// TIA Portal V17 export
// export: Created 2023-12-05T13:40:23.3729222Z, ExportSetting WithDefaults, DisplayName Totally Integrated Automation Portal, DisplayVersion V17, DisplayName TIA Portal Openness, DisplayVersion V17, DisplayName TIA Portal Version Control Interface, DisplayVersion V17, DisplayName SINAMICS Startdrive Advanced, DisplayVersion V17, DisplayName SINAMICS Startdrive G130, G150, S120, S150, SINAMICS MV, S210, DisplayVersion V17, DisplayName SINAMICS Startdrive G110M, G120, G120C, G120D, G120P, G115D, DisplayVersion V17, DisplayName STEP 7 Professional, DisplayVersion V17, DisplayName STEP 7 Safety, DisplayVersion V17, DisplayName WinCC Professional, DisplayVersion V17
DATA_BLOCK "ALARMS"   // DB70
{ S7_Optimized_Access := 'FALSE' }
VERSION : 0.1
// stored: AutoNumber false, DBAccessibleFromOPCUA true, DBAccessibleFromWebserver true, IsOnlyStoredInLoadMemory false, IsWriteProtectedInAS false
   VAR RETAIN
      GENERAL : Struct
         MESSAGES : Struct
            ST1 : Struct
               SwitchNotInAuto : Bool;   // ST100 Not in AUTO MODE
               TakeOutFromST1 : Bool;   // ST100 Take out tank
               "ST1OP02+ST1OP03BoxAlmostFull" : Bool;   // ST1 Punchings Box almost full
               ST1OP04BoxAlmostFull : Bool;   // ST1OP04 FSU Box almost full
               "ST1OP05+ST1OP06+ST1OP07BoxAlmostFull" : Bool;   // ST1OP05+OP06+OP07 Box almost full
               RemoveST1OP08Grip : Bool;   // Remove Component From Gripper ST1OP08
               RemoveST1OP09Grip : Bool;   // Remove Component From Gripper ST1OP09
               RemoveST1OP10Grip : Bool;   // Remove Component From Gripper ST1OP10
               SetupST1 : Bool;   // SETUP MODE ST100
               EngageDoor : Bool;   // Engage Door
               RemoveTankST1 : Bool;   // ST100 Remove Tank
               LoadTankST1 : Bool;   // ST100 Load Tank
               RemoveTankBadST1 : Bool;   // ST100 Remove BAD Tank
               RemoveTankDoubtfullST1 : Bool;   // ST100 Remove DOUBTFULL Tank
               LoadST1OP08ComponentToGripper : Bool;   // Load component ST1OP08 to gripper
               LoadST1OP09ComponentToGripper : Bool;   // Load component ST1OP09 to gripper
               LoadST1OP10ComponentToGripper : Bool;   // Load component ST1OP10 to gripper
               StartToStart : Bool;   // ST100 Press Start Cycle to Start Cycle
               ControlON : Bool;   // Press Control ON to Turn ON Safety Relay
               SwitchAuto : Bool;   // Switch ST100 to AUTO
               ConfBasicGen : Bool;   // Press GENRAL Start Cycle to Initiate Basic Position
               BasicGen : Bool;   // Press GENRAL Basic Push Button to Basic Position
               ConfBasicST1 : Bool;   // ST100 Press Start Cycle to Initiate Basic Position
               BasicST1 : Bool;   // ST100 Press Basic Push Button to Basic Position
               msgStartReworkSt100 : Bool;   // ST100 Press Start Cycle to start Rework Mode
               CycleNotFinST1 : Bool;   // ST100 Cycle not Finish(Make REWORK or Press Start Cycle for BAD TANK)
               "Weekend mode activated" : Bool;   // Weekend mode activated
               msgSelectOPRewSt100 : Bool;   // ST100 Select operation in REWORK MODE
               InFootST1OP10HA : Bool;   // Footprint heating all ST1OP10
               InFootST1OP08MA : Bool;   // Footprint matching all ST1OP08
               InFootST1OP09HT : Bool;   // Footprint heating tank ST1OP09
               InFootST1OP10MA : Bool;   // Footprint matching all ST1OP10
               InFootST1OP09HA : Bool;   // Footprint heating all ST1OP09
               InFootST1OP09MT : Bool;   // Footprint matching tank ST1OP09
               InFootST1OP08HT : Bool;   // Footprint heating tank ST1OP08
               InFootST1OP09MA : Bool;   // Footprint matching all ST1OP09
               InFootST1OP08HA : Bool;   // Footprint heating all ST1OP08
               InFootST1OP08MT : Bool;   // Footprint matching tank ST1OP08
               InFootST1OP10HT : Bool;   // Footprint heating tank ST1OP10
               InFootST1OP10MT : Bool;   // Footprint matching tank ST1OP10
               ST1OP08CriticalValue : Bool;   // ST1OP08 Component critical value
               ResetAlmST1 : Bool;
               ST1OP10CriticalValue : Bool;   // ST1OP10 Component critical value
               ST1OP09CriticalValue : Bool;   // ST1OP09 Component critical value
               ST1OP05KnifeAlmostUsed : Bool;   // ST1OP05 Knife almost used
               ST1OP04KnifeAlmostUsed : Bool;   // ST1OP04 Knife almost used
               ST1OP07KnifeAlmostUsed : Bool;   // ST1OP07 Knife almost used
               ST1OP06KnifeAlmostUsed : Bool;   // ST1OP06 Knife almost used
               OperatorScannerOFF : Bool;   // Operator Scanner OFF
               EP1 : Bool;   // Error proofing need to be done
               EP2 : Bool;   // Error proofing
               EP3 : Bool;   // Error proofing
               EP4 : Bool;   // Error proofing
               EP5 : Bool;   // Error proofing
               EP6 : Bool;   // Error proofing
               EP7 : Bool;   // Error proofing
               EP8 : Bool;   // Error proofing
               EP9 : Bool;   // Error proofing
               EP10 : Bool;   // Error proofing
               EP11 : Bool;   // Error proofing
               EP12 : Bool;   // Error proofing
               EP13 : Bool;   // Error proofing
               EP14 : Bool;   // Error proofing
               EP15 : Bool;   // Error proofing
               EP16 : Bool;   // Error proofing
               ResetReminders : Bool;   // Reset reminders
               InhBarcode1 : Bool;   // Inhibition barcode scanner ST1
               InhBarcode2 : Bool;
               EngageCurtain : Bool;   // Press Start cycle to engage Lightcurtain on ST1
               spare_3 : Bool;
               spare_4 : Bool;
               spare_5 : Bool;
               spare_6 : Bool;
               spare_7 : Bool;
               spare_8 : Bool;
               spare_9 : Bool;
               spare_10 : Bool;
               spare_11 : Bool;
               spare_12 : Bool;
               spare_13 : Bool;
            END_STRUCT;
            ST2 : Struct
               SwitchNotInAuto : Bool;   // ST200 Not in AUTO MODE
               "ST2OP02+ST2OP05BoxAlmostFull" : Bool;   // ST2OP02 + ST2OP05 Box almost full
               EngageDoor : Bool;   // Engage Door
               SetupST2 : Bool;   // SETUP MODE ST200
               RemoveST2OP04Grip : Bool;   // Remove Component From Gripper ST2OP04
               RemoveST2OP06Grip : Bool;   // Remove Component From Gripper ST2OP06
               LoadTankST2 : Bool;   // ST100 Load Tank
               RemoveTankST2 : Bool;   // ST100 Remove Tank
               RemoveTankBadST2 : Bool;   // ST100 Remove BAD Tank
               RemoveTankDoubtfullST2 : Bool;   // ST100 Remove DOUBTFULL Tank
               LoadST2OP06ComponentToGripper : Bool;   // Load component ST2OP06 to gripper
               LoadST2OP04ComponentToGripper : Bool;   // Load component ST2OP04 to gripper
               StartToStart : Bool;   // ST100 Press Start Cycle to Start Cycle
               SwitchAuto : Bool;   // Switch ST200 to AUTO
               ConfBasicST2 : Bool;   // ST200 Press Start Cycle to Initiate Basic Position
               BasicST2 : Bool;   // ST200 Press Basic Push Button to Basic Position
               msgSelectOPRewSt200 : Bool;   // ST200 Select operation in REWORK MODE
               CycleNotFinST2 : Bool;   // ST200 Cycle not Finish(Make REWORK or Press Start Cycle for BAD TANK)
               ResetAlmST2 : Bool;
               msgStartReworkSt200 : Bool;   // ST200 Press Start Cycle to start Rework Mode
               InFootST2OP04MA : Bool;   // Footprint matching all ST2OP04
               InFootST2OP06HT : Bool;   // Footprint heating tank ST2OP06
               InFootST2OP04MT : Bool;   // Footprint matching tank ST2OP04
               InFootST2OP04HA : Bool;   // Footprint heating all ST2OP04
               InFootST2OP06MA : Bool;   // Footprint matching all ST2OP06
               InFootST2OP04HT : Bool;   // Footprint heating tank ST2OP04
               InFootST2OP06MT : Bool;   // Footprint matching tank ST2OP06
               InFootST2OP06HA : Bool;   // Footprint heating all ST2OP06
               ST2OP04CriticalValue : Bool;   // ST2OP04 Component critical value
               ST2OP06CriticalValue : Bool;   // ST2OP06 Component critical value
               EP1 : Bool;   // Error proofing need to be done
               EP2 : Bool;   // Error proofing
               EP3 : Bool;   // Error proofing
               EP4 : Bool;   // Error proofing
               EP5 : Bool;   // Error proofing
               EP6 : Bool;   // Error proofing
               EP7 : Bool;   // Error proofing
               EP8 : Bool;   // Error proofing
               EP9 : Bool;   // Error proofing
               EP10 : Bool;   // Error proofing
               EP11 : Bool;   // Error proofing
               EP12 : Bool;   // Error proofing
               EP13 : Bool;   // Error proofing
               EP14 : Bool;   // Error proofing
               EP15 : Bool;   // Error proofing
               EP16 : Bool;   // Error proofing
               ST2OP02KnifeAlmostUsed : Bool;   // ST2OP02 Knife almost used
               ST2OP05KnifeAlmostUsed : Bool;   // ST2OP05 Knife almost used
               ResetReminders : Bool;   // Reset reminders
               InhBarcode1 : Bool;   // Inhibition barcode scanner ST2
               InhBarcode2 : Bool;
               EngageCurtain : Bool;   // Press start cycle to engage lightcurtain on ST2
               spare_3 : Bool;
               spare_4 : Bool;
               spare_5 : Bool;
               spare_6 : Bool;
               spare_7 : Bool;
               spare_8 : Bool;
               spare_9 : Bool;
               spare_10 : Bool;
               spare_11 : Bool;
               spare_12 : Bool;
               spare_13 : Bool;
               spare_14 : Bool;
               spare_15 : Bool;
               spare_16 : Bool;
               spare_17 : Bool;
               spare_18 : Bool;
               spare_19 : Bool;
               spare_20 : Bool;
               spare_21 : Bool;
               spare_22 : Bool;
               spare_23 : Bool;
               spare_24 : Bool;
               spare_25 : Bool;
               spare_26 : Bool;
               spare_27 : Bool;
               spare_28 : Bool;
               spare_29 : Bool;
               spare_30 : Bool;
            END_STRUCT;
            ST3 : Struct
               SwitchNotInAuto : Bool;   // ST300 Not in AUTO MODE
               EngageDoor : Bool;   // Engage Door
               SetupST3 : Bool;   // SETUP MODE ST300
               RemoveST3OP02Grip : Bool;   // Remove Component From Gripper ST3OP02
               RemoveST3OP03Grip : Bool;   // Remove Component From Gripper ST3OP03
               RemoveST3OP04Grip : Bool;   // Remove Component From Gripper ST3OP04
               RemoveST3OP05Grip : Bool;   // Remove Component From Gripper ST3OP05
               LoadTankST3 : Bool;   // ST100 Load Tank
               RemoveTankST3 : Bool;   // ST100 Remove Tank
               RemoveTankBadST3 : Bool;   // ST100 Remove BAD Tank
               RemoveTankDoubtfullST3 : Bool;   // ST100 Remove DOUBTFULL Tank
               LoadST3OP02ComponentToGripper : Bool;   // Load component ST3OP02 to gripper
               LoadST3OP03ComponentToGripper : Bool;   // Load component ST3OP03 to gripper
               LoadST3OP04ComponentToGripper : Bool;   // Load component ST3OP04 to gripper
               LoadST3OP05ComponentToGripper : Bool;   // Load component ST3OP05 to gripper
               StartToStart : Bool;   // ST100 Press Start Cycle to Start Cycle
               SwitchAuto : Bool;   // Switch ST300 to AUTO
               ConfBasicST3 : Bool;   // ST300 Press Start Cycle to Initiate Basic Position
               BasicST3 : Bool;   // ST300 Press Basic Push Button to Basic Position
               CycleNotFinST3 : Bool;   // ST300 Cycle not Finish(Make REWORK or Press Start Cycle for BAD TANK)
               msgStartReworkSt300 : Bool;   // ST300 Press Start Cycle to start Rework Mode
               msgSelectOPRewSt300 : Bool;   // ST300 Select operation in REWORK MODE
               spare_13 : Bool;
               ResetAlmST3 : Bool;
               InFootST3OP02HA : Bool := false;   // Footprint heating all ST3OP02
               InFootST3OP02MA : Bool := false;   // Footprint matching all ST3OP02
               InFootST3OP02HT : Bool := false;   // Footprint heating tank ST3OP02
               InFootST3OP02MT : Bool := false;   // Footprint matching tank ST3OP02
               InFootST3OP03HA : Bool;   // Footprint heating all ST3OP03
               InFootST3OP03MA : Bool;   // Footprint matching all ST3OP03
               InFootST3OP03HT : Bool;   // Footprint heating tank ST3OP03
               InFootST3OP03MT : Bool;   // Footprint matching tank ST3OP03
               InFootST3OP04HA : Bool := false;   // Footprint heating all ST3OP04
               InFootST3OP04MA : Bool := false;   // Footprint matching all ST3OP04
               InFootST3OP04HT : Bool := false;   // Footprint heating tank ST3OP04
               InFootST3OP04MT : Bool := false;   // Footprint matching tank ST3OP04
               InFootST3OP05HA : Bool := false;   // Footprint heating all ST3OP05
               InFootST3OP05MA : Bool := false;   // Footprint matching all ST3OP05
               InFootST3OP05HT : Bool := false;   // Footprint heating tank ST3OP05
               InFootST3OP05MT : Bool := false;   // Footprint matching tank ST3OP05
               ST3OP03CriticalValue : Bool;   // ST3OP03 Component critical value
               ST3OP02CriticalValue : Bool;   // ST3OP02 Component critical value
               ST3OP05CriticalValue : Bool;   // ST3OP05 Component critical value
               ST3OP04CriticalValue : Bool;   // ST3OP04 Component critical value
               EP2 : Bool;   // Error proofing
               EP1 : Bool;   // Error proofing need to be done
               EP4 : Bool;   // Error proofing
               EP3 : Bool;   // Error proofing
               EP6 : Bool;   // Error proofing
               EP5 : Bool;   // Error proofing
               EP8 : Bool;   // Error proofing
               EP7 : Bool;   // Error proofing
               EP10 : Bool;   // Error proofing
               EP9 : Bool;   // Error proofing
               EP12 : Bool;   // Error proofing
               EP11 : Bool;   // Error proofing
               EP14 : Bool;   // Error proofing
               EP13 : Bool;   // Error proofing
               EP16 : Bool;   // Error proofing
               EP15 : Bool;   // Error proofing
               ResetReminders : Bool;   // Reset reminders
               InhBarcode1 : Bool;   // Inhibition barcode scanner ST3
               InhBarcode2 : Bool;
               EngageCurtain : Bool;   // Press start cycle to engage lightcurtain on ST3
               spare_3 : Bool;
               spare_4 : Bool;
               spare_5 : Bool;
               spare_6 : Bool;
               spare_7 : Bool;
               spare_8 : Bool;
               spare_9 : Bool;
               spare_10 : Bool;
               spare_11 : Bool;
               spare_12 : Bool;
               spare_14 : Bool;
               spare_15 : Bool;
               spare_16 : Bool;
               spare_17 : Bool;
               spare_18 : Bool;
               spare_19 : Bool;
            END_STRUCT;
            ST4 : Struct
               SwitchNotInAuto : Bool;   // ST400 Not in AUTO MODE
               "ST4OP02+ST4OP03BoxAlmostFull" : Bool;   // ST4 PUNCHINGS BOX
               EngageDoor : Bool;   // Engage Door
               SetupST4 : Bool;   // SETUP MODE ST400
               RemoveST4OP05Grip : Bool;   // Remove Component From Gripper ST4OP05
               RemoveST4OP04Grip : Bool;   // Remove Component From Gripper ST4OP04
               RemoveST4OP07Grip : Bool;   // Remove Component From Gripper ST4OP07
               RemoveST4OP08Grip : Bool;   // Remove Component From Gripper ST4OP08
               RemoveST4OP06Grip : Bool;   // Remove Component From Gripper ST4OP06
               LoadTankST4 : Bool;   // ST100 Load Tank
               RemoveTankST4 : Bool;   // ST100 Remove Tank
               RemoveTankDoubtfullST4 : Bool;   // ST100 Remove DOUBTFULL Tank
               RemoveTankBadST4 : Bool;   // ST100 Remove BAD Tank
               LoadST4OP04ComponentToGripper : Bool;   // Load component ST4OP04 to gripper
               LoadST4OP05ComponentToGripper : Bool;   // Load component ST4OP05 to gripper
               LoadST4OP08ComponentToGripper : Bool;   // Load component ST4OP08 to gripper
               LoadST4OP07ComponentToGripper : Bool;   // Load component ST4OP07 to gripper
               LoadST4OP06ComponentToGripper : Bool;   // Load component ST4OP06 to gripper
               StartToStart : Bool;   // ST100 Press Start Cycle to Start Cycle
               SwitchAuto : Bool;   // Switch ST400 to AUTO
               BasicST4 : Bool;   // ST400 Press Basic Push Button to Basic Position
               ConfBasicST4 : Bool;   // ST400 Press Start Cycle to Initiate Basic Position
               CycleNotFinST4 : Bool;   // ST400 Cycle not Finish(Make REWORK or Press Start Cycle for BAD TANK)
               msgStartReworkSt400 : Bool;   // ST400 Press Start Cycle to start Rework Mode
               msgSelectOPRewSt400 : Bool;   // ST400 Select operation in REWORK MODE
               ResetAlmST4 : Bool;
               InFootST4OP04MA : Bool := false;   // Footprint matching all ST4OP04
               InFootST4OP04HA : Bool := false;   // Footprint heating all ST4OP04
               InFootST4OP04MT : Bool := false;   // Footprint matching tank ST4OP04
               InFootST4OP04HT : Bool := false;   // Footprint heating tank ST4OP04
               InFootST4OP05MA : Bool;   // Footprint matching all ST4OP05
               InFootST4OP05HA : Bool;   // Footprint heating all ST4OP05
               InFootST4OP05MT : Bool;   // Footprint matching tank ST4OP05
               InFootST4OP05HT : Bool;   // Footprint heating tank ST4OP05
               InFootST4OP06MA : Bool;   // Footprint matching all ST4OP06
               InFootST4OP06HA : Bool;   // Footprint heating all ST4OP06
               InFootST4OP06MT : Bool;   // Footprint matching tank ST4OP06
               InFootST4OP06HT : Bool;   // Footprint heating tank ST4OP06
               InFootST4OP07MA : Bool;   // Footprint matching all ST4OP07
               InFootST4OP07HA : Bool;   // Footprint heating all ST4OP07
               InFootST4OP07MT : Bool;   // Footprint matching tank ST4OP07
               InFootST4OP07HT : Bool;   // Footprint heating tank ST4OP07
               InFootST4OP08MA : Bool;   // Footprint matching all ST4OP08
               InFootST4OP08HA : Bool;   // Footprint heating all ST4OP08
               InFootST4OP08MT : Bool;   // Footprint matching tank ST4OP08
               InFootST4OP08HT : Bool;   // Footprint heating tank ST4OP08
               ST4OP05CriticalValue : Bool;   // ST4OP05 Component critical value
               ST4OP04CriticalValue : Bool;   // ST4OP04 Component critical value
               ST4OP07CriticalValue : Bool;   // ST4OP07 Component critical value
               ST4OP06CriticalValue : Bool;   // ST4OP06 Component critical value
               ST4OP08CriticalValue : Bool;   // ST4OP08 Component critical value
               EP2 : Bool;   // Error proofing
               EP1 : Bool;   // Error proofing need to be done
               EP4 : Bool;   // Error proofing
               EP3 : Bool;   // Error proofing
               EP6 : Bool;   // Error proofing
               EP5 : Bool;   // Error proofing
               EP8 : Bool;   // Error proofing
               EP7 : Bool;   // Error proofing
               EP10 : Bool;   // Error proofing
               EP9 : Bool;   // Error proofing
               EP12 : Bool;   // Error proofing
               EP11 : Bool;   // Error proofing
               EP14 : Bool;   // Error proofing
               EP13 : Bool;   // Error proofing
               EP16 : Bool;   // Error proofing
               EP15 : Bool;   // Error proofing
               ResetReminders : Bool;   // Reset reminders
               InhBarcode1 : Bool;   // Inhibition barcode scanner ST4
               InhBarcode2 : Bool;
               EngageCurtain : Bool;   // Press start cycle to engage lightcurtain on ST4
               spare_3 : Bool;
               spare_4 : Bool;
               spare_5 : Bool;
               spare_6 : Bool;
               spare_7 : Bool;
               spare_8 : Bool;
               spare_9 : Bool;
               spare_10 : Bool;
               spare_11 : Bool;
            END_STRUCT;
            Temp3 : Array[40..69] of Byte;
         END_STRUCT;
         UnitsCycleTimeExceeded : Struct
            msgST1OP02 : Bool;   // Cycle time exceeded - ST1OP02
            msgST1OP03 : Bool;   // Cycle time exceeded - ST1OP03
            msgST1OP04 : Bool;   // Cycle time exceeded - ST1OP04
            msgST1OP05 : Bool;   // Cycle time exceeded - ST1OP05
            msgST1OP06 : Bool;   // Cycle time exceeded - ST1OP06
            msgST1OP07 : Bool;   // Cycle time exceeded - ST1OP07
            msgST1OP08 : Bool;   // Cycle time exceeded - ST1OP08
            msgST1OP09 : Bool;   // Cycle time exceeded - ST1OP09
            msgST1OP10 : Bool;   // Cycle time exceeded - ST1OP10
            msgST2OP02 : Bool;   // Cycle time exceeded - ST2OP02
            msgST2OP03 : Bool;   // Cycle time exceeded - ST2OP03
            msgST2OP04 : Bool;   // Cycle time exceeded - ST2OP04
            msgST2OP05 : Bool;   // Cycle time exceeded - ST2OP05
            msgST2OP06 : Bool;   // Cycle time exceeded - ST2OP06
            msgST3OP02 : Bool;   // Cycle time exceeded - ST3OP02
            msgST3OP03 : Bool;   // Cycle time exceeded - ST3OP03
            msgST3OP04 : Bool;   // Cycle time exceeded - ST3OP04
            msgST3OP05 : Bool;   // Cycle time exceeded - ST3OP05
            msgST4OP02 : Bool;   // Cycle time exceeded - ST4OP02
            msgST4OP03 : Bool;   // Cycle time exceeded - ST4OP03
            msgST4OP04 : Bool;   // Cycle time exceeded - ST4OP04
            msgST4OP05 : Bool;   // Cycle time exceeded - ST4OP05
            msgST4OP06 : Bool;   // Cycle time exceeded - ST4OP06
            msgST4OP07 : Bool;   // Cycle time exceeded - ST4OP07
            msgST4OP08 : Bool;   // Cycle time exceeded - ST4OP08
            msgSpare_2_5 : Bool;
            msgSpare_2_6 : Bool;
            msgSpare_2_7 : Bool;
            msgSpare_3_0 : Bool;
            msgSpare_3_1 : Bool;
            msgSpare_3_2 : Bool;
            msgSpare_3_3 : Bool;
            msgSpare_3_4 : Bool;
            msgSpare_3_5 : Bool;
            msgSpare_3_6 : Bool;
            msgSpare_3_7 : Bool;
            Temp1 : Array[4..7] of Byte;
         END_STRUCT;
         UnitsInAuto_Messages : Struct
            msgST1OP02 : Bool;   // Waiting for inteverntion - ST1OP02 in auto
            msgST1OP03 : Bool;   // Waiting for inteverntion - ST1OP03 in auto
            msgST1OP04 : Bool;   // Waiting for inteverntion - ST1OP04 in auto
            msgST1OP05 : Bool;   // Waiting for inteverntion - ST1OP05 in auto
            msgST1OP06 : Bool;   // Waiting for inteverntion - ST1OP06 in auto
            msgST1OP07 : Bool;   // Waiting for inteverntion - ST1OP07 in auto
            msgST1OP08 : Bool;   // Waiting for inteverntion - ST1OP08 in auto
            msgST1OP09 : Bool;   // Waiting for inteverntion - ST1OP09 in auto
            msgST1OP10 : Bool;   // Waiting for inteverntion - ST1OP10 in auto
            msgST2OP02 : Bool;   // Waiting for inteverntion - ST2OP02 in auto
            msgST2OP03 : Bool;   // Waiting for inteverntion - ST2OP03 in auto
            msgST2OP04 : Bool;   // Waiting for inteverntion - ST2OP04 in auto
            msgST2OP05 : Bool;   // Waiting for inteverntion - ST2OP05 in auto
            msgST2OP06 : Bool;   // Waiting for inteverntion - ST2OP06 in auto
            msgSpare_0_5 : Bool;
            msgSpare_0_6 : Bool;
            msgSpare_0_7 : Bool;
            spare : Bool;
            msgST3OP02 : Bool;   // Waiting for inteverntion - ST3OP02 in auto
            msgST3OP03 : Bool;   // Waiting for inteverntion - ST3OP03 in auto
            msgST3OP04 : Bool;   // Waiting for inteverntion - ST3OP04 in auto
            msgST3OP05 : Bool;   // Waiting for inteverntion - ST3OP05 in auto
            spare_2 : Bool;
            msgSpare_1_2 : Bool;
            msgSpare_1_3 : Bool;
            msgSpare_1_4 : Bool;
            msgSpare_1_5 : Bool;
            msgSpare_1_6 : Bool;
            msgSpare_1_7 : Bool;
            spare_3 : Bool;
            msgST4OP02 : Bool;   // Waiting for inteverntion - ST4OP02 in auto
            msgST4OP03 : Bool;   // Waiting for inteverntion - ST4OP03 in auto
            msgST4OP04 : Bool;   // Waiting for inteverntion - ST4OP04 in auto
            msgST4OP05 : Bool;   // Waiting for inteverntion - ST4OP05 in auto
            msgST4OP06 : Bool;   // Waiting for inteverntion - ST4OP06 in auto
            msgST4OP07 : Bool;   // Waiting for inteverntion - ST4OP07 in auto
            msgST4OP08 : Bool;   // Waiting for inteverntion - ST4OP08 in auto
            spare_1 : Bool;
            msgSpare_2_7 : Bool;
            msgSpare_3_0 : Bool;
            msgSpare_3_1 : Bool;
            msgSpare_3_2 : Bool;
            msgSpare_3_3 : Bool;
            msgSpare_3_4 : Bool;
            msgSpare_3_5 : Bool;
            msgSpare_3_6 : Bool;
            msgSpare_3_7 : Bool;
            Temp1 : Array[4..7] of Byte;
         END_STRUCT;
         MovingUnits_Messages : Struct
            msgST1Base : Bool;   // Waiting for inteverntion - ST100 Base is moving
            "msgCommonTransfer102+103" : Bool;   // Waiting for inteverntion - ST4OP04+OP06+OP07 is moving
            "msgCommonTransfer105+106" : Bool;   // Waiting for inteverntion - ST4OP04+OP06+OP07 is moving
            msgST1OP02 : Bool;   // Waiting for inteverntion - ST4OP04+OP06+OP07 is moving
            msgST1OP03 : Bool;   // Waiting for inteverntion - ST4OP04+OP06+OP07 is moving
            msgST1OP04 : Bool;   // Waiting for inteverntion - ST4OP04+OP06+OP07 is moving
            msgST1OP05 : Bool;   // Waiting for inteverntion - ST4OP04+OP06+OP07 is moving
            msgST1OP06 : Bool;   // Waiting for inteverntion - ST4OP04+OP06+OP07 is moving
            msgST1OP07 : Bool;   // Waiting for inteverntion - ST4OP04+OP06+OP07 is moving
            msgST1OP08 : Bool;   // Waiting for inteverntion - ST4OP04+OP06+OP07 is moving
            msgST1OP09 : Bool;   // Waiting for inteverntion - ST4OP04+OP06+OP07 is moving
            msgST1OP10 : Bool;   // Waiting for inteverntion - ST4OP04+OP06+OP07 is moving
            msgST1OP11 : Bool;   // Waiting for inteverntion - ST4OP09 (BOWL FEEDER) is moving
            msgST2Base : Bool;   // Waiting for inteverntion - ST200 Base is moving
            msgST2OP02 : Bool;   // Waiting for inteverntion - ST2OP02 (CUT ROV) is moving
            msgST2OP03 : Bool;   // Waiting for inteverntion - ST2OP03 (CUT NIPPLE E5) is moving
            msgST2OP04 : Bool;   // Waiting for inteverntion - ST2OP03 (CUT NIPPLE E5) is moving
            msgST2OP05 : Bool;   // Waiting for inteverntion - ST2OP03 (CUT NIPPLE E5) is moving
            msgST2OP06 : Bool;   // Waiting for inteverntion - ST2OP03 (CUT NIPPLE E5) is moving
            msgST2OP11 : Bool;   // Waiting for inteverntion - ST4OP09 (BOWL FEEDER) is moving
            msgST3Base : Bool;   // Waiting for inteverntion - ST300 Base is moving
            msgST3OP02 : Bool;   // Waiting for inteverntion - ST2OP07 (CUT NIPPLE L8) is moving
            msgST3OP03 : Bool;   // Waiting for inteverntion - ST3OP03 (WELD ROV) is moving
            msgST3OP04 : Bool;   // Waiting for inteverntion - ST3OP04 (WELD HSB1) is moving
            msgST3OP05 : Bool;   // Waiting for inteverntion - ST3OP07 (WELD ROV CFLVV) is moving
            msgST3OP07 : Bool;   // Waiting for inteverntion - ST4OP09 (BOWL FEEDER) is moving
            msgST4Base : Bool;   // Waiting for inteverntion - ST400 Base is moving
            "msgCommonTransfer404+405" : Bool;   // Waiting for inteverntion - ST4OP02+OP03+OP05 is moving
            "msgCommonTransfer402+403" : Bool;   // Waiting for inteverntion - ST2OP03 + ST2OP07 Tr Horizontal is moving
            msgST4OP01 : Bool;   // Waiting for inteverntion - ST4OP01 (WELD NIPPLE) is moving
            msgST4OP02 : Bool;   // Waiting for inteverntion - ST4OP02 (WELD CLIP 1) is moving
            msgST4OP03 : Bool;   // Waiting for inteverntion - ST4OP03 (WELD CLIP 2) is moving
            msgST4OP04 : Bool;   // Waiting for inteverntion - ST4OP04 (WELD CLIP 3) is moving
            msgST4OP05 : Bool;   // Waiting for inteverntion - ST4OP05 (WELD CLIP 4) is moving
            msgST4OP06 : Bool;   // Waiting for inteverntion - ST4OP06 (WELD CLIP 5) is moving
            msgST4OP07 : Bool;   // Waiting for inteverntion - ST4OP07 (WELD CLIP 6) is moving
            msgST4OP08 : Bool;   // Waiting for inteverntion - ST4OP09 (BOWL FEEDER) is moving
            msgST4OP10 : Bool;   // Waiting for inteverntion - ST4OP09 (BOWL FEEDER) is moving
            msgSpare_3_1 : Bool;
            msgSpare_2_2 : Bool;
            msgSpare_3_3 : Bool;
            msgInterventionST1 : Bool;   // INTERVENTION ST1
            msgInterventionST2 : Bool;   // INTERVENTION ST2
            msgInterventionST3 : Bool;   // INTERVENTION ST3
            msgInterventionST4 : Bool;   // INTERVENTION ST4
            msgSpare_1_4 : Bool;
            spare_3 : Bool;
            spare_4 : Bool;
            "msgDoorST100BACK#1" : Bool;   // ST1 Door Back #1 Open I21.3 / B156.12
            "msgDoorST100BACK#2" : Bool;   // ST1 Door Back #2 Open I21.4 / B157.12
            msgDoorST200 : Bool;   // ST2 Door Open I23.3 / B256.12
            msgDoorST300 : Bool;   // ST3 Door Open I4.3 / B357.12
            msgDoorST400 : Bool;   // ST4 Door Open I6.3 / B456.12
            msgSpare_1 : Bool;
            msgSpare_4_6 : Bool;
            msgSpare_4_7 : Bool;
            Temp1 : Array[6..7] of Byte;
         END_STRUCT;
         GENERAL_ALARMS : Struct
            ESTOP_Control_Cabinet : Bool;   // Emergency Stop Control Cabinet I0.1 / S22.2
            ESTOP_ST1_ACP : Bool;   // Emergency Stop ST 1 ACP I21.6 / S154.5
            ESTOP_ST1_MCP : Bool;   // Emergency Stop ST 1 MCP I22.0 / S155.5
            ESTOP_ST1_DOOR : Bool;   // Emergency Stop ST 1 Door I21.0 / S156.4
            ESTOP_HMI : Bool;   // Emergency Stop HMI I20.0 / S257.5
            ESTOP_ST2_MCP : Bool;   // Emergency Stop ST 2 MCP I24.0 / S255.5
            spare_1 : Bool;
            ESTOP_ST2_DOOR : Bool;   // Emergency Stop ST 2 Door I23.0 / S256.4
            ESTOP_ST3_MCP : Bool;   // Emergency Stop ST 3 MCP I5.0 / S356.5
            spare_2 : Bool;
            ESTOP_ST3_DOOR : Bool;   // Emergency Stop ST 3 Door I4.0 / S357.4
            ESTOP_ST4_MCP : Bool;   // Emergency Stop ST 4 MCP I7.0 / S455.5
            ESTOP_ST4_ACP : Bool;   // Emergency Stop ST 4 ACP I6.6 / S454.5
            ESTOP_ST4_DOOR : Bool;   // Emergency Stop ST 4 Door I6.0 / S456.4
            Spare0_7 : Bool;
            Spare1_0 : Bool;
            Spare1_1 : Bool;
            ConnectionEKI_Alm : Bool;   // Badge Scanner not connected
            OperatorNotLoggedAlm : Bool;   // Operator Not Logged
            Spare1_4 : Bool;
            Spare1_5 : Bool;
            Spare1_6 : Bool;
            NeedToChangeover : Bool;
            Spare2_0 : Bool;
            Spare2_1 : Bool;
            Spare2_2 : Bool;
            FingerPrintAccess : Bool;   // Finger print without any access
            Spare2_4 : Bool;
            Spare2_6 : Bool;
            Spare2_7 : Bool;
            AirPressLow : Bool;   // Air presure too low I0.4 / K16.5
            AirPressLowMV : Bool;   // Air presure too low after MAIN VALVE I0.5 / K16.10
            MainPressValve1 : Bool;   // Main pressure station valve 1 NO OK I0.4 / K16.5
            MainPressValve2 : Bool;   // Main pressure station valve 2 NO OK I0.5 / K16.10
            PahseControl : Bool;   // Fault Phase Control Not OK I0.3 / K2.5
            ElectricBoxTemp : Bool;   // Fault Main Electric Box temperature too high I0.2 / B56.7
            Spare3_7 : Bool;
            Spare4_2 : Bool;
            Spare4_3 : Bool;
            Spare4_4 : Bool;
            Spare4_5 : Bool;
            Spare4_6 : Bool;
            Spare4_7 : Bool;
            "ST1OP08-ST1OP10BatchFifo" : Bool;
            ST2OP04BatchFifo : Bool;
            ST2OP06BatchFifo : Bool;
            ST3OP02BatchFifo : Bool;
            ST3OP03BatchFifo : Bool;
            ST3OP04BatchFifo : Bool;
            ST3OP05BatchFifo : Bool;
            "ST4OP04-ST4OP05BatchFifo" : Bool;
            "ST4OP06-ST4OP08BatchFifo" : Bool;
            "ST1OP08-ST1OP10Block" : Bool;
            ST2OP04Block : Bool;
            ST2OP06Block : Bool;
            ST3OP02Block : Bool;
            ST3OP03Block : Bool;
            ST3OP04Block : Bool;
            ST3OP05Block : Bool;
            "ST4OP04-ST4OP05Block" : Bool;
            "ST4OP06-ST4OP08Block" : Bool;
            Spare6_0 : Bool;
            Spare6_1 : Bool;
            Spare6_2 : Bool;
            Spare6_4 : Bool;
            Spare6_5 : Bool;
            Spare6_6 : Bool;
            Spare6_7 : Bool;
            Spare7_0 : Bool;
            Spare7_1 : Bool;
            Spare7_2 : Bool;
            Spare7_3 : Bool;
            Spare7_4 : Bool;
            Spare7_5 : Bool;
            Spare7_6 : Bool;
            Spare7_7 : Bool;
            Spare11_7 : Bool;
            Temp1 : Array[8..87] of Byte;
         END_STRUCT;
         NODES_ALARMS : Struct
            N1Alm : Bool;
            N2Alm : Bool;
            N3Alm : Bool;
            N4Alm : Bool;   // Node nr 4 ET200 Main Electric Box not responding
            N5Alm : Bool;   // Node nr 5 ET200 A1 Electric Box not responding
            N6Alm : Bool;   // Node nr 6 WEISS Inverter not responding
            N7Alm : Bool;
            N8Alm : Bool;   // Node nr 8 EKI
            N9Alm : Bool;
            N10Alm : Bool;   // Node nr 10 ABB Cabinet
            N11Alm : Bool;   // Node nr 11 CPX DP11 not responding
            N12Alm : Bool;   // Node nr 12 CPX DP12 not responding
            N13Alm : Bool;   // Node nr 13 CPX DP13 not responding
            N14Alm : Bool;   // Node nr 14 CPX DP14 not responding
            N15Alm : Bool;
            N16Alm : Bool;
            N17Alm : Bool;
            N18Alm : Bool;
            N19Alm : Bool;
            N20Alm : Bool;
            N21Alm : Bool;   // Node nr 21 CPX DP21 not responding
            N22Alm : Bool;   // Node nr 22 CPX DP22 not responding
            N23Alm : Bool;
            N24Alm : Bool;
            N25Alm : Bool;
            N26Alm : Bool;
            N27Alm : Bool;
            N28Alm : Bool;
            N29Alm : Bool;
            N30Alm : Bool;
            N31Alm : Bool;   // Node nr 31 CPX DP31 not responding
            N32Alm : Bool;   // Node nr 32 CPX DP32 not responding
            N33Alm : Bool;   // Node nr 33 CPX DP33 not responding
            N34Alm : Bool;
            N35Alm : Bool;
            N36Alm : Bool;
            N37Alm : Bool;
            N38Alm : Bool;
            N39Alm : Bool;
            N40Alm : Bool;
            N41Alm : Bool;   // Node nr 41 CPX DP41 not responding
            N42Alm : Bool;   // Node nr 42 CPX DP42 not responding
            N43Alm : Bool;   // Node nr 43 CPX DP43 not responding
            N44Alm : Bool;
            N45Alm : Bool;
            N46Alm : Bool;
            N47Alm : Bool;
            N48Alm : Bool;
            N49Alm : Bool;
            N50Alm : Bool;
            N51Alm : Bool;
            N52Alm : Bool;
            N53Alm : Bool;
            N54Alm : Bool;
            N55Alm : Bool;   // Node nr 55 ABB Robot not responding
            N56Alm : Bool;   // Node nr 56 Weiss Table not responding
            N57Alm : Bool;
            N58Alm : Bool;
            N59Alm : Bool;
            N60Alm : Bool;
            N61Alm : Bool;
            N62Alm : Bool;
            N63Alm : Bool;
            N250Alm : Bool;
            Temp1 : Array[8..9] of Byte;
         END_STRUCT;
      END_STRUCT;
      ST1 : Struct
         GENERAL : Struct   // ST1 GENERAL
            TankBAD : Bool;   // Tank BAD after Manual Mode
            VerCrossed : Bool;   // ST1 Vertical light curtain crossed without authorization
            HorCrossed : Bool;   // ST1 Horizontal light curtain crossed without authorization
            VerNotEngaged : Bool;   // ST1 Cannot engage vertical light curtain
            HorNotEngaged : Bool;   // ST1 Cannot engage horizontal light curtain
            VerActive : Bool;   // ST1 Vertical light curtain not active
            HorActive : Bool;   // ST1 Horizontal light curtain not active
            TankAbsent_FOTO : Bool;   // ST1 Tank absent on foto I101.2/B175.8
            Tank_TempOutOfTol : Bool;   // Tank temperature out of tolerance PIW500 / B190.3
            Tank_TempSensBrok : Bool;   // Tank temperature sensor broken PIW500 / B190.3
            SqlST1 : Bool;   // ST2 SQL Trigger not reseted after 10s
            SqlST2 : Bool;   // ST3 SQL Trigger not reseted after 10s
            SqlST3 : Bool;   // ST4 SQL Trigger not reseted after 10s
            SqlST4 : Bool;   // ST1 SQL Trigger not reseted after 10s
            TankAbsent_ISOPIN_L : Bool;   // ST1 Tank absent on ISOPIN Left I100.0/B174.4
            TankAbsent_ISOPIN_R : Bool;   // ST1 Tank absent on ISOPIN Right I100.1/B174.6
            BarcodeTankNotRead : Bool;   // Alarm Tank barcode not read
            BarcodeTankNotCorrect : Bool;   // Alarm Tank barcode not correct with selected version
            FIFO_Tank : Bool;   // FIFO Alarm - Tank was processed
            Spare2_3 : Bool;
            BarcodeTankNotRead2 : Bool;   // Alarm Tank barcode 2not read
            BarcodeTankNotCorrect2 : Bool;   // Alarm Tank barcode2 not correct with selected version
            FIFO_Tank2 : Bool;   // FIFO Alarm 2- Tank was processed
            Spare2_7 : Bool;
            NoReleaseToStart : Bool;   // No release authorization from Traceability for Station 1 start cycle. Please acknowledge.
            NoReleaseToUnclamp : Bool;   // No release authorization from Traceability for Station 1 unclamp Tank. Please acknowledge.
            WaitReletoStAlmRes : Bool;   // Traceability for Station 1 is waiting for release to start alarm reset
            WaitResultReadAlmRes : Bool;   // Traceability for Station 1 is waiting for result read alarm reset
            TraceTrigON : Bool;   // Station 1 Traceability log fault (trigger still ON)
            Spare3_5 : Bool;
            Spare3_6 : Bool;
            Spare3_7 : Bool;
            TableDobulPos : Bool;
            TableInvertNotEn : Bool;   // Fault Tank temperature out of tolerance
            TablerInvNotReady : Bool;   // Fault Tank temperature sensor broken
            TableNotInPos : Bool;   // Empty the slug bin ST1OP1/ST1OP2
            TableTime : Bool;
            TablePosRun : Bool;
            TableSafety : Bool;
            TableSumEr : Bool;   // ST1OP01 CUT FSU Slug not detected frame I120.4/B157.10
            TableSumWar : Bool;   // ST1OP02 CUT ICV Slug not detected frame I120.3/B157.12
            Spare5_1 : Bool;
            Spare5_2 : Bool;
            ST1PunchingBoxFull : Bool;   // ST1 Left Slug box full
            spare_1 : Bool;
            Spare5_5 : Bool;
            Spare5_6 : Bool;
            Spare5_7 : Bool;
            Spare : Array[6..9] of Byte;
         END_STRUCT;
         BASE : Struct   // SHUTTER
            ClampDownWP : Bool;   // ST1 Base Clamp down failed to advance I100.2/B174.8
            ClampDownPP : Bool;   // ST1 Base Clamp down failed to reverse I100.3/B174.10
            ClampDownBS : Bool;   // ST1 Base Clamp down both sensors ON I100.2-3/B174.8-10
            MobileBaseWP : Bool;   // ST1 Base Mobile base failed to advance I100.4/B174.12
            MobileBasePP : Bool;   // ST1 Base Mobile base failed to reverse I100.5/B174.14
            MobileBaseTS : Bool;   // ST1 Base Mobile base both sensors ON I100.4-5/B174.12-14
            ClampUpLeftWP : Bool;   // ST1 Base Clamp up left failed to advance I100.6/B174.16
            ClampUpLeftPP : Bool;   // ST1 Base Clamp up left failed to reverse I100.7/B174.18
            ClampUpLeftBS : Bool;   // ST1 Base Clamp up left both sensors ON I100.2-3/B174.16-18
            ClampUpRightWP : Bool;   // ST1 Base Clamp up right failed to advance I101.0/B175.4
            ClampUpRightPP : Bool;   // ST1 Base Clamp up right failed to reverse I101.1/B175.6
            ClampUpRightBS : Bool;   // ST1 Base Clamp up right both sensors ON I100.0-1/B175.4-6
            Temp1 : Array[2..9] of Byte;
         END_STRUCT;
         ST1OP02 : Struct   // PUNCHING 1
            TrHorAdvFlt : Bool;   // ST1OP02 (PUNCHING 1) Tr Horizontal Failed To Advance I120.6,I121.6/B176.16,B177.8
            TrHorRetFlt : Bool;   // ST1OP02 (PUNCHING 1) Tr Horizontal Failed To Reverse I120.7/B176.18
            TrHorTSFlt : Bool;   // ST1OP02 (PUNCHING 1) Tr Horizontal both sensor ON I120.6-7,I121.6/B176.16-18,B177.8
            StampAdvFlt : Bool;   // ST1OP02 (PUNCHING 1) Stamp Failed To Advance I120.0/B176.4
            StampRevFlt : Bool;   // ST1OP02 (PUNCHING 1) Stamp Failed To Reverse I120.1/B176.6
            StampTSFlt : Bool;   // ST1OP02 (PUNCHING 1) Stamp both sensor ON I120.0-1/B176.4-6
            OperationNotCompletedCorrectlyFlt : Bool;   // ST1OP02 (PUNCHING 1) Operation not completed correctly RC1601
            SlugDetectionFlt : Bool;   // ST1OP02 (PUNCHING 1) Slug Detection on Frame Fault I101.4/B175.12 RC1600
            SlugStillPresent : Bool;   // ST1OP02 (PUNCHING 1) Slug stuck in blowing system I121.6/B177.16
            CycleNotStarted : Bool;   // ST1OP02 (PUNCHING 1) Cycle Not Started
            CycleNotFinished : Bool;   // ST1OP02 (PUNCHING 1) Cycle Not Finished
            CycleTime : Bool;   // ST1OP02 (PUNCHING 1) Cycle Time too long
            Presence : Bool;   // ST1OP02 (PUNCHING 1) Alarm Presence
            CarriageHorizontalWP : Bool;   // ST1OP02 (PUNCHING 1) Carriage Horizontal Failed To Advance I120.2/B176.8
            CarriageHorizontalPP : Bool;   // ST1OP02 (PUNCHING 1) Carriage Horizontal Failed To Reverse I120.3/B176.10
            CarriageHorizontalBS : Bool;   // ST1OP02 (PUNCHING 1) Carriage Horizontal both sensor ON I120.2-3/B176.8-10
            CarriageVerticalWP : Bool;   // ST1OP02 (PUNCHING 1) Carriage Vertical Failed To Advance I120.4/B176.12
            CarriageVerticalPP : Bool;   // ST1OP02 (PUNCHING 1) Carriage Vertical Failed To Reverse I120.5/B176.14
            CarriageVerticalBS : Bool;   // ST1OP02 (PUNCHING 1) Carriage Vertical both sensor ON I120.4-5/B176.12-14
            BumperTrHorizWP : Bool;   // ST1OP02 (PUNCHING 1) Bumper Tr Horizontal Failed To Advance I121.0/B177.4
            BumperTrHorizPP : Bool;   // ST1OP02 (PUNCHING 1) Bumper Tr Horizontal Failed To Reverse I121.1/B177.6
            BumperTrHorizBS : Bool;   // ST1OP02 (PUNCHING 1) Bumper Tr Horizontal both sensor ON I121.0-1/B177.4-6
            Temp1 : Array[6..11] of Byte;
         END_STRUCT;
         ST1OP03 : Struct   // PUNCHING 2
            TrHorAdvFlt : Bool;   // ST1OP03 (PUNCHING 2) Tr Horizontal Failed To Advance I130.6,I131.2/B178.16,B179.8
            TrHorRetFlt : Bool;   // ST1OP03 (PUNCHING 2) Tr Horizontal Failed To Reverse I130.7/B178.18
            TrHorTSFlt : Bool;   // ST1OP03 (PUNCHING 2) Tr Horizontal both sensor ON I130.6-7,I131.6/B178.16-18,B179.8
            StampAdvFlt : Bool;   // ST1OP03 (PUNCHING 2) Stamp Failed To Advance I130.0/B178.4
            StampRevFlt : Bool;   // ST1OP03 (PUNCHING 2) Stamp Failed To Reverse I130.1/B178.6
            StampTSFlt : Bool;   // ST1OP03 (PUNCHING 2) Stamp both sensor ON I130.0-1/B178.4-6
            OperationNotCompletedCorrectlyFlt : Bool;   // ST1OP03 (PUNCHING 2) Operation not completed correctly RC1601
            SlugDetectionFlt : Bool;   // ST1OP03 (PUNCHING 2) Slug Detection on Frame Fault I101.4/B175.12 RC1600
            SlugStillPresent : Bool;   // ST1OP03 (PUNCHING 2) Slug stuck in blowing system I131.6/B179.16
            CycleNotStarted : Bool;   // ST1OP03 (PUNCHING 2) Cycle Not Started
            CycleNotFinished : Bool;   // ST1OP03 (PUNCHING 2) Cycle Not Finished
            CycleTime : Bool;   // ST1OP03 (PUNCHING 2) Cycle Time too long
            Presence : Bool;   // ST1OP03 (PUNCHING 2) Alarm Presence
            CarriageHorizontalWP : Bool;   // ST1OP03 (PUNCHING 2) Carriage Horizontal Failed To Advance I130.2/B178.8
            CarriageHorizontalPP : Bool;   // ST1OP03 (PUNCHING 2) Carriage Horizontal Failed To Reverse I130.3/B178.10
            CarriageHorizontalBS : Bool;   // ST1OP03 (PUNCHING 2) Carriage Horizontal both sensor ON I130.2-3/B178.8-10
            CarriageVerticalWP : Bool;   // ST1OP03 (PUNCHING 2) Carriage Vertical Failed To Advance I130.4/B178.12
            CarriageVerticalPP : Bool;   // ST1OP03 (PUNCHING 2) Carriage Vertical Failed To Reverse I130.5/B178.14
            CarriageVerticalBS : Bool;   // ST1OP03 (PUNCHING 2) Carriage Vertical both sensor ON I130.4-5/B178.12-14
            BumperTrHorizWP : Bool;   // ST1OP03 (PUNCHING 2) Bumper Tr Horizontal Failed To Advance I131.0/B179.4
            BumperTrHorizPP : Bool;   // ST1OP03 (PUNCHING 2) Bumper Tr Horizontal Failed To Reverse I131.1/B179.6
            BumperTrHorizBS : Bool;   // ST1OP03 (PUNCHING 2) Bumper Tr Horizontal both sensor ON I131.0-1/B179.4-6
            Temp1 : Array[6..11] of Byte;
         END_STRUCT;
         ST1OP04 : Struct   // CUT FSU HV
            UnitTransferAdvFlt : Bool;   // ST1OP04 (Cut FSU HV) Unit Transfer Failed To Advance I140.0/B185.4
            UnitTransferRetFlt : Bool;   // ST1OP04 (Cut FSU HV) Unit Transfer Failed To Return I140.1/B185.6
            UnitTransferTSFlt : Bool;   // ST1OP04 (Cut FSU HV) Unit Transfer Two Sensors ON I140.0-1/B185.4-6
            CuttingAdvFlt : Bool;   // ST1OP04 (Cut FSU HV) Cutting Cylinder Failed To Advance I140.2/B185.8
            CuttingRevFlt : Bool;   // ST1OP04 (Cut FSU HV) Cutting Cylinder Failed To Return I140.3/B185.10
            CuttingTSFlt : Bool;   // ST1OP04 (Cut FSU HV) Cutting Cylinder Two Sensors ON I140.2-3/B185.8-10
            ClampAdvFlt : Bool;   // ST1OP04 (Cut FSU HV) Ring Clamp Failed To Advance I140.4/B185.12
            ClampRevFlt : Bool;   // ST1OP04 (Cut FSU HV) Ring Clamp Failed To Return I140.5/B185.14
            ClampTSFlt : Bool;   // ST1OP04 (Cut FSU HV) Ring Clamp Two Sensors ON I140.4-5/B185.12-14
            FingersAdvFlt : Bool;   // ST1OP04 (Cut FSU HV) Fingers Failed To Advance I140.6/B185.16
            FingersRevFlt : Bool;   // ST1OP04 (Cut FSU HV) Fingers Failed To Return I140.6/B185.16
            FingersTSFlt : Bool;
            Spare1_4Alm : Bool;
            Spare1_5Alm : Bool;
            Spare1_6Alm : Bool;
            Spare1_7Alm : Bool;
            SlugUnitFlt : Bool;   // ST1OP04 (Cut FSU HV) Slug Not Detected on Unit RC300 I140.7/B185.18
            CuttingTimeOutFlt : Bool;   // ST1OP04 (Cut FSU HV) Cutting Time Exceeded RC301
            CylFaultDuringCycleFlt : Bool;   // ST1OP04 (Cut FSU HV) Cylinder Fault During Cycle RC302
            CycleNotFinishFlt : Bool;   // ST1OP04 (Cut FSU HV) Cycle Failed To Finish RC303
            CycleNotStartedFlt : Bool;   // ST1OP04 (Cut FSU HV) Cycle Not Started Fault RC304
            SlugFrameFlt : Bool;   // ST1OP04 (Cut FSU HV) Slug Not Detected by Frame RC305 I101.3/B175.10
            CylPositionLostFlt : Bool;   // ST1OP04 (Cut FSU HV) Cylinders Position Lost in manual RC306
            Spare2_7Alm : Bool;
            Spare3_0Alm : Bool;
            Spare3_1Alm : Bool;
            Spare3_2Alm : Bool;
            Spare3_3Alm : Bool;
            Spare3_4Alm : Bool;
            Spare3_5Alm : Bool;
            Spare3_6Alm : Bool;
            Spare3_7Alm : Bool;
            CircuitBreakerTripFlt : Bool;   // ST1OP04 (Cut FSU HV) Circuit Breaker Tripped I25.0/F109.3
            SlugSensorOffFlt : Bool;   // ST1OP04 (Cut FSU HV) Slug sensor OFF I140.7/B185.18
            ContactorOffFlt : Bool;   // ST1OP04 (Cut FSU HV) Motor Contactor OFF I25.1/K144.3
            ContactorOnFlt : Bool;   // ST1OP04 (Cut FSU HV) Motor Contactor ON I25.1/K144.3
            FrameConstantlyONFlt : Bool;   // ST1OP04 (Cut FSU HV) Frame Constanly ON I101.3/B175.10
            ChangeKnife : Bool;   // ST1OP04 (Cut FSU HV) Change knife
            Spare4_6Alm : Bool;
            Spare4_7Alm : Bool;
            CarStopWPAlm : Bool;   // ST1OP04 (Cut FSU HV) Carriage stopper failed to advance I141.0/B186.4
            CarStopPPAlm : Bool;   // ST1OP04 (Cut FSU HV) Carriage stopper failed to reverse I141.1/B186.6
            CarStopBSAlm : Bool;   // ST1OP04 (Cut FSU HV) Carriage stopper both sensors ON I141.0-1/B186.4-6
            TrHorWPAlm : Bool;   // ST1OP04 (Cut FSU HV) Tr horizontal failed to advance I141.2/B186.8
            TrHorPPAlm : Bool;   // ST1OP04 (Cut FSU HV) Tr horizontal failed to reverse I141.3/B186.10
            TrHorBSAlm : Bool;   // ST1OP04 (Cut FSU HV) Tr horizontal both sensors ON I141.2-3/B186.8-10
            Spare5_6Alm : Bool;
            SlugBoxFull : Bool;   // ST1OP04 (Cut FSU HV) Slug box full I242.4 / B266.12
            Temp1 : Array[6..9] of Byte;
         END_STRUCT;
         ST1OP05 : Struct   // CUT ICV HV
            UnitTransferAdvFlt : Bool;   // ST1OP05 (CUT ICV HV) Unit Transfer Failed To Advance I150.0/B194.4
            UnitTransferRetFlt : Bool;   // ST1OP05 (CUT ICV HV) Unit Transfer Failed To Return I150.1/B194.6
            UnitTransferTSFlt : Bool;   // ST1OP05 (CUT ICV HV) Unit Transfer Two Sensors ON I150.0-1/B194.4-6
            CuttingAdvFlt : Bool;   // ST1OP05 (CUT ICV HV) Cutting Cylinder Failed To Advance I150.2/B194.8
            CuttingRevFlt : Bool;   // ST1OP05 (CUT ICV HV) Cutting Cylinder Failed To Return I150.3/B194.10
            CuttingTSFlt : Bool;   // ST1OP05 (CUT ICV HV) Cutting Cylinder Two Sensors ON I150.2-3/B194.8-10
            NeedleAdvFlt : Bool;   // ST1OP05 (CUT ICV HV) Slug Needle Failed To Advance I150.4/B194.12
            NeedleRevFlt : Bool;   // ST1OP05 (CUT ICV HV) Slug Needle Failed To Return I150.5/B194.14
            NeedleTSFlt : Bool;   // ST1OP05 (CUT ICV HV) Slug Needle Two Sensors ON I150.4-5/B194.12-14
            SpareCylFaults : Int;
            SlugUnitFlt : Bool;   // ST1OP05 (CUT ICV HV) Slug Not Detected on Unit RC350 I150.6/B194.16
            CuttingTimeOutFlt : Bool;   // ST1OP05 (CUT ICV HV) Cutting Time Exceeded RC351
            CylFaultDuringCycleFlt : Bool;   // ST1OP05 (CUT ICV HV) Cylinder Fault During Cycle RC352
            CycleNotFinishFlt : Bool;   // ST1OP05 (CUT ICV HV) Cycle Failed To Finish RC353
            CycleNotStartedFlt : Bool;   // ST1OP05 (CUT ICV HV) Cycle Not Started Fault RC354
            SlugFrameFlt : Bool;   // ST1OP05 (CUT ICV HV) Slug Not Detected by Frame RC355 I101.5/B175.14
            ManualUsedFlt : Bool;   // ST1OP05 (CUT ICV HV) Cylinders Position Lost in manual RC356
            Spare2_7Alm : Bool;
            Spare3_0Alm : Bool;
            spare : Bool;
            spare_1 : Bool;
            spare_2 : Bool;
            Spare_8_7Alm : Bool;
            MissingStartFromSTDBlock : Bool;   // ST1OP05 (CUT ICV HV) Missing Start Cycle From Standard Block
            SlugBoxFull : Bool;   // ST1OP05 (CUT ICV HV) + ST1OP06 (CUT ICV CONV) + ST1OP07 (CUT NIPPLE CONV) Slug box full
            Spare3_7Alm : Bool;
            CircuitBreakerTripFlt : Bool;   // ST1OP05 (CUT ICV HV) Circuit Breaker Tripped I25.2/F109.7
            SlugSensorOnFlt : Bool;   // ST1OP05 (CUT ICV HV) Slug sensor ON I150.6/B194.16
            ContactorOffFlt : Bool;   // ST1OP05 (CUT ICV HV) Motor Contactor OFF I25.3/BK144.5
            ContactorOnFlt : Bool;   // ST1OP05 (CUT ICV HV) Motor Contactor ON I25.3/BK144.5
            FrameConstantlyONFlt : Bool;   // ST1OP05 (CUT ICV HV) Frame Constanly ON I101.5/B175.14
            ChangeKnife : Bool;   // ST1OP05 (CUT ICV HV) Change knife
            Spare4_6Alm : Bool;
            Spare4_7Alm : Bool;
            CarStopWPAlm : Bool;   // ST1OP05 (CUT ICV HV) Carriage stopper failed to advance I151.0/B195.4
            CarStopPPAlm : Bool;   // ST1OP05 (CUT ICV HV) Carriage stopper failed to reverse I151.1/B195.6
            CarStopBSAlm : Bool;   // ST1OP05 (CUT ICV HV) Carriage stopper both sensors on I151.0-1/B195.6
            HorizontalTrAdvFlt : Bool;   // ST1OP05 (CUT ICV HV) + ST1OP06 (CUT ICV HV) Transfer Horizontal failed to advance I151.2/B195.8
            HorizontalTrRetFlt : Bool;   // ST1OP05 (CUT ICV HV) + ST1OP06 (CUT ICV HV) Transfer Horizontal failed to reverse I151.3/B195.10
            HorizontalTrTSFlt : Bool;   // ST1OP05 (CUT ICV HV) + ST1OP06 (CUT ICV HV) Transfer Horizontal both sensors ON I151.2-3 /B195.8-10
            Spare7_6Alm : Bool;
            Spare7_7Alm : Bool;
            Spare8_0Alm : Bool;
            BumperHorizontalTrAdvFlt : Bool;   // ST1OP05 (CUT ICV HV) + ST1OP06 (CUT ICV HV) Bumper Transfer Horizontal failed to advance I151.4/B195.12
            BumperHorizontalTrRetFlt : Bool;   // ST1OP05 (CUT ICV HV) + ST1OP06 (CUT ICV HV) Bumper Transfer Horizontal failed to reverse I151.6/B195.14
            BumperHorizontalTrTSFlt : Bool;   // ST1OP05 (CUT ICV HV) + ST1OP06 (CUT ICV HV) Bumper Transfer Horizontal both sensors ON I151.4-6/B195.12-14
            Spare7_6Alm_2 : Bool;
            Spare7_7Alm_2 : Bool;
            Spare8_0Alm_2 : Bool;
            VacuumFlapWP : Bool;
            VacuumFlapPP : Bool;
            VacuumFlapBS : Bool;
            Spare7_6Alm_4 : Bool;
            Spare7_7Alm_4 : Bool;
            Spare8_0Alm_4 : Bool;
            Spare8_0Alm_5 : Bool;
            Spare8_0Alm_6 : Bool;
            Spare8_0Alm_7 : Bool;
         END_STRUCT;
         ST1OP06 : Struct   // CUT ICV CONV
            UnitTransferAdvFlt : Bool;   // ST1OP06 (CUT ICV CONV) Unit Transfer Failed To Advance I160.0/B196.4
            UnitTransferRetFlt : Bool;   // ST1OP06 (CUT ICV CONV) Unit Transfer Failed To Return I160.1/B196.6
            UnitTransferTSFlt : Bool;   // ST1OP06 (CUT ICV CONV) Unit Transfer Two Sensors ON I160.0-1/B196.4-6
            CuttingAdvFlt : Bool;   // ST1OP06 (CUT ICV CONV) Cutting Cylinder Failed To Advance I160.2/B196.8
            CuttingRevFlt : Bool;   // ST1OP06 (CUT ICV CONV) Cutting Cylinder Failed To Return I160.3/B196.10
            CuttingTSFlt : Bool;   // ST1OP06 (CUT ICV CONV) Cutting Cylinder Two Sensors ON I160.2-3/B196.8-10
            NeedleAdvFlt : Bool;   // ST1OP06 (CUT ICV CONV) Slug Needle Failed To Advance I160.4/B196.12
            NeedleRevFlt : Bool;   // ST1OP06 (CUT ICV CONV) Slug Needle Failed To Return I160.5/B196.14
            NeedleTSFlt : Bool;   // ST1OP06 (CUT ICV CONV) Slug Needle Two Sensors ON I160.4-5/B196.12-14
            SpareCylFaults : Int;
            SlugUnitFlt : Bool;   // ST1OP06 (CUT ICV CONV) Slug Not Detected on Unit RC350 I160.6/B196.16
            CuttingTimeOutFlt : Bool;   // ST1OP06 (CUT ICV CONV) Cutting Time Exceeded RC351
            CylFaultDuringCycleFlt : Bool;   // ST1OP06 (CUT ICV CONV) Cylinder Fault During Cycle RC352
            CycleNotFinishFlt : Bool;   // ST1OP06 (CUT ICV CONV) Cycle Failed To Finish RC353
            CycleNotStartedFlt : Bool;   // ST1OP06 (CUT ICV CONV) Cycle Not Started Fault RC354
            SlugFrameFlt : Bool;   // ST1OP06 (CUT ICV CONV) Slug Not Detected by Frame RC355 I101.5/B175.14
            ManualUsedFlt : Bool;   // ST1OP06 (CUT ICV CONV) Cylinders Position Lost in manual RC356
            Spare2_7Alm : Bool;
            Spare3_0Alm : Bool;
            BumperHorizontalWPAlm : Bool;
            BumperHorizontalPPAlm : Bool;
            BumperHorizontalBSAlm : Bool;
            Spare_8_7Alm : Bool;
            MissingStartFromSTDBlock : Bool;   // ST1OP06 (CUT ICV CONV) Missing Start Cycle From Standard Block
            SlugBoxFull : Bool;
            Spare3_7Alm : Bool;
            CircuitBreakerTripFlt : Bool;   // ST1OP06 (CUT ICV CONV) Circuit Breaker Tripped I25.4/F109.11
            SlugSensorOnFlt : Bool;   // ST1OP06 (CUT ICV CONV) Slug sensor ON I160.6/B196.16
            ContactorOffFlt : Bool;   // ST1OP06 (CUT ICV CONV) Motor Contactor OFF I25.5/K144.7
            ContactorOnFlt : Bool;   // ST1OP06 (CUT ICV CONV) Motor Contactor ON I25.5/K144.7
            FrameConstantlyONFlt : Bool;   // ST1OP06 (CUT ICV CONV) Frame Constanly ON I101.5/B175.14
            ChangeKnife : Bool;   // ST1OP06 (CUT ICV CONV) Change knife
            Spare4_6Alm : Bool;
            Spare4_7Alm : Bool;
            CarStopWPAlm : Bool;   // ST1OP06 (CUT ICV CONV) Carriage stopper failed to advance I161.0/B197.4
            CarStopPPAlm : Bool;   // ST1OP06 (CUT ICV CONV) Carriage stopper failed to reverse I161.1/B197.6
            CarStopBSAlm : Bool;   // ST1OP06 (CUT ICV CONV) Carriage stopper both sensors on I161.0-1/B197.4-6
            HorizontalTrAdvFlt : Bool;
            HorizontalTrRetFlt : Bool;
            HorizontalTrTSFlt : Bool;
            Spare7_6Alm : Bool;
            Spare7_7Alm : Bool;
            Spare8_0Alm : Bool;
            VacuumFlapWP : Bool;
            VacuumFlapPP : Bool;
            VacuumFlapBS : Bool;
            Spare7_6Alm_2 : Bool;
            Spare7_7Alm_2 : Bool;
            Spare8_0Alm_2 : Bool;
            Spare7_6Alm_3 : Bool;
            Spare7_7Alm_3 : Bool;
            Spare8_0Alm_3 : Bool;
            Spare7_6Alm_4 : Bool;
            Spare7_7Alm_4 : Bool;
            Spare8_0Alm_4 : Bool;
            Spare8_0Alm_5 : Bool;
            Spare8_0Alm_6 : Bool;
            Spare8_0Alm_7 : Bool;
         END_STRUCT;
         ST1OP07 : Struct   // CUT NIPPLE CONV
            UnitTransferAdvFlt : Bool;   // ST1OP07 (CUT NIPPLE CONV) Unit Transfer Failed To Advance I170.0/B187.4
            UnitTransferRetFlt : Bool;   // ST1OP07 (CUT NIPPLE CONV) Unit Transfer Failed To Return I170.1/B187.6
            UnitTransferTSFlt : Bool;   // ST1OP07 (CUT NIPPLE CONV) Unit Transfer Two Sensors ON I170.0-1/B187.4-6
            CuttingAdvFlt : Bool;   // ST1OP07 (CUT NIPPLE CONV) Cutting Cylinder Failed To Advance I170.2/B187.8
            CuttingRevFlt : Bool;   // ST1OP07 (CUT NIPPLE CONV) Cutting Cylinder Failed To Return I170.3/B187.10
            CuttingTSFlt : Bool;   // ST1OP07 (CUT NIPPLE CONV) Cutting Cylinder Two Sensors ON I170.2-3/B187.8-10
            NeedleAdvFlt : Bool;   // ST1OP07 (CUT NIPPLE CONV) Slug Needle Failed To Advance I170.4/B187.12
            NeedleRevFlt : Bool;   // ST1OP07 (CUT NIPPLE CONV) Slug Needle Failed To Return I170.5/B187.14
            NeedleTSFlt : Bool;   // ST1OP07 (CUT NIPPLE CONV) Slug Needle Two Sensors ON I170.4-5/B187.12-14
            SpareCylFaults : Int;
            SlugUnitFlt : Bool;   // ST1OP07 (CUT NIPPLE CONV) Slug Not Detected on Unit RC350 I170.6/B187.16
            CuttingTimeOutFlt : Bool;   // ST1OP07 (CUT NIPPLE CONV) Cutting Time Exceeded RC351
            CylFaultDuringCycleFlt : Bool;   // ST1OP07 (CUT NIPPLE CONV) Cylinder Fault During Cycle RC352
            CycleNotFinishFlt : Bool;   // ST1OP07 (CUT NIPPLE CONV) Cycle Failed To Finish RC353
            CycleNotStartedFlt : Bool;   // ST1OP07 (CUT NIPPLE CONV) Cycle Not Started Fault RC354
            SlugFrameFlt : Bool;   // ST1OP07 (CUT NIPPLE CONV) Slug Not Detected by Frame RC355 I101.5/B175.14
            ManualUsedFlt : Bool;   // ST1OP07 (CUT NIPPLE CONV) Cylinders Position Lost in manual RC356
            Spare2_7Alm : Bool;
            Spare3_0Alm : Bool;
            BumperHorizontalWPAlm : Bool;
            BumperHorizontalPPAlm : Bool;
            BumperHorizontalBSAlm : Bool;
            Spare_8_7Alm : Bool;
            MissingStartFromSTDBlock : Bool;   // ST1OP07 (CUT NIPPLE CONV) Missing Start Cycle From Standard Block
            SlugBoxFull : Bool;
            Spare3_7Alm : Bool;
            CircuitBreakerTripFlt : Bool;   // ST1OP07 (CUT NIPPLE CONV) Circuit Breaker Tripped I25.6/F109.15
            SlugSensorOnFlt : Bool;   // ST1OP07 (CUT NIPPLE CONV) Slug sensor ON I170.6/B187.16
            ContactorOffFlt : Bool;   // ST1OP07 (CUT NIPPLE CONV) Motor Contactor OFF I25.7/K144.9
            ContactorOnFlt : Bool;   // ST1OP07 (CUT NIPPLE CONV) Motor Contactor ON I25.7/K144.9
            FrameConstantlyONFlt : Bool;   // ST1OP07 (CUT NIPPLE CONV) Frame Constanly ON I101.5/B175.14
            ChangeKnife : Bool;   // ST1OP07 (CUT NIPPLE CONV) Change knife
            Spare4_6Alm : Bool;
            Spare4_7Alm : Bool;
            CarStopWPAlm : Bool;   // ST1OP07 (CUT NIPPLE CONV) Carriage stopper failed to advance I171.0/B188.4
            CarStopPPAlm : Bool;   // ST1OP07 (CUT NIPPLE CONV) Carriage stopper failed to reverse I171.1/B188.6
            CarStopBSAlm : Bool;   // ST1OP07 (CUT NIPPLE CONV) Carriage stopper both sensors on I171.0-1/B188.4-6
            CrossTrAdvFlt : Bool;   // ST1OP07 (CUT NIPPLE CONV) Transfer Cross failed to advance I171.2/B188.8
            CrossTrRetFlt : Bool;   // ST1OP07 (CUT NIPPLE CONV) Transfer Cross failed to reverse I171.3/B188.10
            CrossTrTSFlt : Bool;   // ST1OP07 (CUT NIPPLE CONV) Transfer Cross both sensors ON I171.2-3/188.8-10
            Spare7_6Alm : Bool;
            Spare7_7Alm : Bool;
            Spare8_0Alm : Bool;
            StopperCrossTrAdvFlt : Bool;   // ST1OP07 (CUT NIPPLE CONV) Stopper Tr Cross failed to advance I171.4/B188.12
            StopperCrossTrRetFlt : Bool;   // ST1OP07 (CUT NIPPLE CONV) Stopper Tr Cross failed to reverse I171.5/B188.14
            StopperCrossTrTSFlt : Bool;   // ST1OP07 (CUT NIPPLE CONV) Stopper Tr Cross both sensors ON I171.4-5/B188.12-14
            Spare7_6Alm_2 : Bool;
            Spare7_7Alm_2 : Bool;
            Spare8_0Alm_2 : Bool;
            VacuumFlapWP : Bool;
            VacuumFlapPP : Bool;
            VacuumFlapBS : Bool;
            Spare7_6Alm_4 : Bool;
            Spare7_7Alm_4 : Bool;
            Spare8_0Alm_4 : Bool;
            Spare8_0Alm_5 : Bool;
            Spare8_0Alm_6 : Bool;
            Spare8_0Alm_7 : Bool;
         END_STRUCT;
         ST1OP08 : Struct   // WELD / WELD HSB1 HV
            HeaterTransferAdvFlt : Bool;   // ST1OP08 (WELD HSB1 HV) Heater Transfer Failed to Advance Ixx.X
            HeaterTransferRetFlt : Bool;   // ST1OP08 (WELD HSB1 HV) Heater Transfer Failed to Return Ixx.X
            HeaterTransferTSFlt : Bool;   // ST1OP08 (WELD HSB1 HV) Heater Transfer Two Sensors on Ixx.X-Ixx.X
            GcylAdvHeatingFlt : Bool;   // ST1OP08 (WELD HSB1 HV) Gcyl Failed to Advance Heating I180.2/B203.8
            GcylAdvCoolingFlt : Bool;   // ST1OP08 (WELD HSB1 HV) Gcyl Failed to Advance Cooling I180.1/B203.6
            GcylAdvLoadingFlt : Bool;   // ST1OP08 (WELD HSB1 HV) Gcyl Failed to Advance Loading I180.0/B203.4
            GcylRetFlt : Bool;   // ST1OP08 (WELD HSB1 HV) Gcyl Failed to Return I180.3/B203.10
            GcylTSFlt : Bool;   // ST1OP08 (WELD HSB1 HV) Gcyl Two Sensors on I180.0/B203.4 - I180.3/B203.10
            HcylAdvFlt : Bool;   // ST1OP08 (WELD HSB1 HV) Hcyl Failed to Advance I180.4/B203.12 (Ret Sensor for BC)
            HcylRevFlt : Bool;   // ST1OP08 (WELD HSB1 HV) Hcyl Failed to Return I180.5/B203.14
            HcylTSFlt : Bool;   // ST1OP08 (WELD HSB1 HV) Hcyl Two Sensors on I180.4/B203.12-I130.5/B203.14
            GripperAdvGripFlt : Bool;   // ST1OP08 (WELD HSB1 HV) Gripper Failed to Grip (Ungrip sensor Fault) I180.6/B203.14
            GripperRetUngripFlt : Bool;   // ST1OP08 (WELD HSB1 HV) Gripper Failed to Ungrip Sensor Fault I180.6/B203.14
            GripTSFlt : Bool;   // not used
            SpareCylFaultsInt0 : Int;
            SpareCylFaultsDInt0 : DInt;
            CompHeatPosFlt : Bool;   // ST1OP08 (WELD HSB1 HV) Component Failed To Gcyl Heating Position I180.2/B203.8 RC201/101
            TankHeatPosFlt : Bool;   // ST1OP08 (WELD HSB1 HV) Hotplate Failed To Hcyl Heating Position I180.4/B203.12 RC217
            CompCoolPosFlt : Bool;   // ST1OP08 (WELD HSB1 HV) Component Failed To Gcyl Cooling Position I180.1/B203.6 RC202/102
            OpenTimeFlt : Bool;   // ST1OP08 (WELD HSB1 HV) Open Time Exceeded RC203/103
            TempDuringCycleFlt : Bool;   // ST1OP08 (WELD HSB1 HV) Hotplate Temperature Fault During Cycle RC204/104
            ReservedRC0_5 : Bool;
            CompHeatPressFlt : Bool;   // ST1OP08 (WELD HSB1 HV) Component Heating Pressure Out Of Tolerance RC205/105
            ReservedRC0_7 : Bool;
            CompCoolPressFlt : Bool;   // ST1OP08 (WELD HSB1 HV) Component Cooling Pressure Out Of Tolerance RC206/106
            ReservedRC1_1 : Bool;
            ReservedRC1_2 : Bool;
            ReservedRC1_3 : Bool;
            ReservedRC1_4 : Bool;
            ReservedRC1_5 : Bool;
            TankHeatPressFlt : Bool;   // ST1OP08 (WELD HSB1 HV) Hcyl Heating Pressure Out Of Tolerance RC207/107
            ReservedRC1_7 : Bool;
            ReservedRC2_0 : Bool;
            ReservedRC2_1 : Bool;
            ReservedRC2_2 : Bool;
            ReservedRC2_3 : Bool;
            CycleNotFinishFlt : Bool;   // ST1OP08 (WELD HSB1 HV) Cycle Failed To Finish RC211/111
            CycleNotStartedFlt : Bool;   // ST1OP08 (WELD HSB1 HV) Cycle Not Started Fault RC212/112
            ReservedRC2_6 : Bool;
            ReservedRC2_7 : Bool;
            ReservedRC3_0 : Bool;
            TankHeatContactFlt : Bool;   // ST1OP08 (WELD HSB1 HV) Tank Heating Contact Pressure Calc Out Of Tolerance RC213/113
            ReservedRC3_2 : Bool;
            ReservedRC3_3 : Bool;
            MeltedComponentFlt : Bool;   // ST1OP08 (WELD HSB1 HV) Remove Melted Component From Gripper I181.0/B204.4 RC214/114
            ReservedRC3_5 : Bool;
            CylFaultDuringCycleFlt : Bool;   // ST1OP08 (WELD HSB1 HV) Cylinder Fault During Cycle RC215/115
            ReservedRC3_7 : Bool;
            ManualUsedFlt : Bool;   // ST1OP08 (WELD HSB1 HV) Manual Movements Used RC216/116
            CompPresent1AfterHeatFlt : Bool;   // ST1OP08 (WELD HSB1 HV) Component Present 1 Missing After Heating I181.0/B204.4 RC208/108
            CompPresent2AfterHeatFlt : Bool;   // ST1OP08 (WELD HSB1 HV) Component Present 2 Missing After Heating Ixx.X RC218/118
            CompPresent3AfterHeatFlt : Bool;   // ST1OP08 (WELD HSB1 HV) Component Present 3 Missing After Heating Ixx.X RC219/119
            CompPresent4AfterHeatFlt : Bool;   // ST1OP08 (WELD HSB1 HV) Component Present 4 Missing After Heating Ixx.X RC220/120
            CompPresent5AfterHeatFlt : Bool;   // ST1OP08 (WELD HSB1 HV) Component Present 5 Missing After Heating Ixx.X RC221/121
            CompPresent6AfterHeatFlt : Bool;   // ST1OP08 (WELD HSB1 HV) Component Present 6 Missing After Heating Ixx.X RC222/122
            CompPresent7AfterHeatFlt : Bool;   // ST1OP08 (WELD HSB1 HV) Component Present 7 Missing After Heating Ixx.X RC223/123
            CompPresent8AfterHeatFlt : Bool;   // ST1OP08 (WELD HSB1 HV) Component Present 8 Missing After Heating Ixx.X RC224/124
            RemoveComponent1Flt : Bool;   // ST1OP08 (WELD HSB1 HV) Remove Component From Gripper (Present 1 after welding) I181.0/B204.4 RC209/109
            RemoveComponent2Flt : Bool;   // ST1OP08 (WELD HSB1 HV) Remove Component From Gripper (Present 2 after welding) Ixx.X RC225/125
            RemoveComponent3Flt : Bool;   // ST1OP08 (WELD HSB1 HV) Remove Component From Gripper (Present 3 after welding) Ixx.X RC226/126
            RemoveComponent4Flt : Bool;   // ST1OP08 (WELD HSB1 HV) Remove Component From Gripper (Present 4 after welding) Ixx.X RC227/127
            RemoveComponent5Flt : Bool;   // ST1OP08 (WELD HSB1 HV) Remove Component From Gripper (Present 5 after welding) Ixx.X RC228/128
            RemoveComponent6Flt : Bool;   // ST1OP08 (WELD HSB1 HV) Remove Component From Gripper (Present 6 after welding) Ixx.X RC229/129
            RemoveComponent7Flt : Bool;   // ST1OP08 (WELD HSB1 HV) Remove Component From Gripper (Present 7 after welding) Ixx.X RC230/130
            RemoveComponent8Flt : Bool;   // ST1OP08 (WELD HSB1 HV) Remove Component From Gripper (Present 8 after welding) Ixx.X RC231/131
            CompMissing1Flt : Bool;   // ST1OP08 (WELD HSB1 HV) Component Present 1 Missing In Gripper I181.0/B204.4 RC210/110
            CompMissing2Flt : Bool;   // ST1OP08 (WELD HSB1 HV) Component Present 2 Missing In Gripper Ixx.X RC232/132
            CompMissing3Flt : Bool;   // ST1OP08 (WELD HSB1 HV) Component Present 3 Missing In Gripper Ixx.X RC233/133
            CompMissing4Flt : Bool;   // ST1OP08 (WELD HSB1 HV) Component Present 4 Missing In Gripper Ixx.X RC234/134
            CompMissing5Flt : Bool;   // ST1OP08 (WELD HSB1 HV) Component Present 5 Missing In Gripper Ixx.X RC235/135
            CompMissing6Flt : Bool;   // ST1OP08 (WELD HSB1 HV) Component Present 6 Missing In Gripper Ixx.X RC236/136
            CompMissing7Flt : Bool;   // ST1OP08 (WELD HSB1 HV) Component Present 7 Missing In Gripper Ixx.X RC237/137
            CompMissing8Flt : Bool;   // ST1OP08 (WELD HSB1 HV) Component Present 8 Missing In Gripper Ixx.X RC238/138
            SpareFaultRC : Byte;
            HotplateTempOutFlt : Bool;   // ST1OP08 (WELD HSB1 HV) Hotplate Temperature Out Of Tolerance
            HotplateTempSensorFlt : Bool;   // ST1OP08 (WELD HSB1 HV) Hotplate Thermocouple Wire Break
            HotplateTempDiffereneceTooBigFlt : Bool;   // ST1OP08 (WELD HSB1 HV) Hotplate Thermocouples Difference Too Big
            Reserved0_3 : Bool;
            Reserved0_4 : Bool;
            Reserved0_5 : Bool;
            CompStuckOnTankFlt : Bool;   // ST1OP08 (WELD HSB1 HV) Component Stuck On Tank Must reset to Ungrip Component
            TempSetFlt : Bool;   // ST1OP08 (WELD HSB1 HV) Hotplate Tempearture Setpoint Out Of Range
            Reserved1_0 : Bool;
            RemoveHeatedComponentFlt : Bool;   // ST1OP08 (WELD HSB1 HV) Remove Heated Component
            CleanHotplatesFlt : Bool;   // ST1OP08 (WELD HSB1 HV) Clean Hotplates
            NoDetectionUsed : Bool;   // ST1OP08 (WELD HSB1 HV) No Detection Used (PLC program issue)
            SpareAlarmsDInt0 : DInt;
            HotTempChanFlt : Bool;   // ST1OP08 (WELD HSB1 HV) Hotplate Temperature is not changing
            Spare_1 : Bool;
            Spare_2 : Bool;
            Spare_3 : Bool;
            Spare_4 : Bool;
            Spare_5 : Bool;
            TrCommonAdvFlt : Bool;
            TrCommonRetFlt : Bool;
            TrCommonTsFlt : Bool;
            Spare_6 : Bool;
            Spare_7 : Bool;
            Spare_8 : Bool;
            TrStopperVerticalWPAlm : Bool;
            TrStopperVerticalPPAlm : Bool;
            TrStopperVerticalBSAlm : Bool;
            Spare_9 : Bool;
            Spare_10 : Bool;
            Spare_11 : Bool;
            LoadingStopperWP : Bool;   // ST1OP08 (WELD HSB1 HV) Loading stopper Failed to Advance I181.3/B204.10
            LoadingStopperPP : Bool;   // ST1OP08 (WELD HSB1 HV) Loading stopper Failed to Return I181.4/B204.12
            LoadingStopperBS : Bool;   // ST1OP08 (WELD HSB1 HV) Loading stopper Two Sensors on I181.3-4/B204.10-12
            Spare_17 : Bool;
            Spare_18 : Bool;
            Spare_19 : Bool;
            Spare_20 : Bool;
            Spare_21 : Bool;
            Spare_22 : Bool;
            Spare_23 : Bool;
            Spare_24 : Bool;
            Spare_25 : Bool;
            Spare_26 : Bool;
            Spare_27 : Bool;
            Spare_28 : Bool;
            Spare_29 : Bool;
            Spare_30 : Bool;
            Spare_31 : Bool;
            Spare_32 : Bool;
            RemCycleNotStartedBADFromPrevStation : Bool;   // RemCycleNotStartedBADFromPrevStation
            Spare_34 : Bool;
         END_STRUCT;
         ST1OP09 : Struct   // WELD / WELD HSB2 HV
            HeaterTransferAdvFlt : Bool;   // ST1OP09 (WELD HSB2 HV) Heater Transfer Failed to Advance Ixx.X
            HeaterTransferRetFlt : Bool;   // ST1OP09 (WELD HSB2 HV) Heater Transfer Failed to Return Ixx.X
            HeaterTransferTSFlt : Bool;   // ST1OP09 (WELD HSB2 HV) Heater Transfer Two Sensors on Ixx.X-Ixx.X
            GcylAdvHeatingFlt : Bool;   // ST1OP09 (WELD HSB2 HV) Gcyl Failed to Advance Heating I190.2/B205.8
            GcylAdvCoolingFlt : Bool;   // ST1OP09 (WELD HSB2 HV) Gcyl Failed to Advance Cooling I190.1/B205.6
            GcylAdvLoadingFlt : Bool;   // ST1OP09 (WELD HSB2 HV) Gcyl Failed to Advance Loading I190.0/B205.4
            GcylRetFlt : Bool;   // ST1OP09 (WELD HSB2 HV) Gcyl Failed to Return I190.3/B205.10
            GcylTSFlt : Bool;   // ST1OP09 (WELD HSB2 HV) Gcyl Two Sensors on I190.0/B205.4 - I190.3/B205.10
            HcylAdvFlt : Bool;   // ST1OP09 (WELD HSB2 HV) Hcyl Failed to Advance I190.4/B205.12 (Ret Sensor for BC)
            HcylRevFlt : Bool;   // ST1OP09 (WELD HSB2 HV) Hcyl Failed to Return I190.5/B205.14
            HcylTSFlt : Bool;   // ST1OP09 (WELD HSB2 HV) Hcyl Two Sensors on I190.4/B205.12-I190.5/B205.14
            GripperAdvGripFlt : Bool;   // ST1OP09 (WELD HSB2 HV) Gripper Failed to Grip (Ungrip sensor Fault) I190.6/B205.16
            GripperRetUngripFlt : Bool;   // ST1OP09 (WELD HSB2 HV) Gripper Failed to Ungrip Sensor Fault I190.6/B205.16
            GripTSFlt : Bool;   // not used
            SpareCylFaultsInt0 : Int;
            SpareCylFaultsDInt0 : DInt;
            CompHeatPosFlt : Bool;   // ST1OP09 (WELD HSB2 HV) Component Failed To Gcyl Heating Position I190.2/B205.8 RC201/101
            TankHeatPosFlt : Bool;   // ST1OP09 (WELD HSB2 HV) Hotplate Failed To Hcyl Heating Position I190.4/B205.12 RC217
            CompCoolPosFlt : Bool;   // ST1OP09 (WELD HSB2 HV) Component Failed To Gcyl Cooling Position I190.1/B205.6 RC202/102
            OpenTimeFlt : Bool;   // ST1OP09 (WELD HSB2 HV) Open Time Exceeded RC203/103
            TempDuringCycleFlt : Bool;   // ST1OP09 (WELD HSB2 HV) Hotplate Temperature Fault During Cycle RC204/104
            ReservedRC0_5 : Bool;
            CompHeatPressFlt : Bool;   // ST1OP09 (WELD HSB2 HV) Component Heating Pressure Out Of Tolerance RC205/105
            ReservedRC0_7 : Bool;
            CompCoolPressFlt : Bool;   // ST1OP09 (WELD HSB2 HV) Component Cooling Pressure Out Of Tolerance RC206/106
            ReservedRC1_1 : Bool;
            ReservedRC1_2 : Bool;
            ReservedRC1_3 : Bool;
            ReservedRC1_4 : Bool;
            ReservedRC1_5 : Bool;
            TankHeatPressFlt : Bool;   // ST1OP09 (WELD HSB2 HV) Hcyl Heating Pressure Out Of Tolerance RC207/107
            ReservedRC1_7 : Bool;
            ReservedRC2_0 : Bool;
            ReservedRC2_1 : Bool;
            ReservedRC2_2 : Bool;
            ReservedRC2_3 : Bool;
            CycleNotFinishFlt : Bool;   // ST1OP09 (WELD HSB2 HV) Cycle Failed To Finish RC211/111
            CycleNotStartedFlt : Bool;   // ST1OP09 (WELD HSB2 HV) Cycle Not Started Fault RC212/112
            ReservedRC2_6 : Bool;
            ReservedRC2_7 : Bool;
            ReservedRC3_0 : Bool;
            TankHeatContactFlt : Bool;   // ST1OP09 (WELD HSB2 HV) Tank Heating Contact Pressure Calc Out Of Tolerance RC213/113
            ReservedRC3_2 : Bool;
            ReservedRC3_3 : Bool;
            MeltedComponentFlt : Bool;   // ST1OP09 (WELD HSB2 HV) Remove Melted Component From Gripper I181.1/B204.6 RC214/114
            ReservedRC3_5 : Bool;
            CylFaultDuringCycleFlt : Bool;   // ST1OP09 (WELD HSB2 HV) Cylinder Fault During Cycle RC215/115
            ReservedRC3_7 : Bool;
            ManualUsedFlt : Bool;   // ST1OP09 (WELD HSB2 HV) Manual Movements Used RC216/116
            CompPresent1AfterHeatFlt : Bool;   // ST1OP09 (WELD HSB2 HV) Component Present 1 Missing After Heating I181.1/B204.6 RC208/108
            CompPresent2AfterHeatFlt : Bool;   // ST1OP09 (WELD HSB2 HV) Component Present 2 Missing After Heating Ixx.X RC218/118
            CompPresent3AfterHeatFlt : Bool;   // ST1OP09 (WELD HSB2 HV) Component Present 3 Missing After Heating Ixx.X RC219/119
            CompPresent4AfterHeatFlt : Bool;   // ST1OP09 (WELD HSB2 HV) Component Present 4 Missing After Heating Ixx.X RC220/120
            CompPresent5AfterHeatFlt : Bool;   // ST1OP09 (WELD HSB2 HV) Component Present 5 Missing After Heating Ixx.X RC221/121
            CompPresent6AfterHeatFlt : Bool;   // ST1OP09 (WELD HSB2 HV) Component Present 6 Missing After Heating Ixx.X RC222/122
            CompPresent7AfterHeatFlt : Bool;   // ST1OP09 (WELD HSB2 HV) Component Present 7 Missing After Heating Ixx.X RC223/123
            CompPresent8AfterHeatFlt : Bool;   // ST1OP09 (WELD HSB2 HV) Component Present 8 Missing After Heating Ixx.X RC224/124
            RemoveComponent1Flt : Bool;   // ST1OP09 (WELD HSB2 HV) Remove Component From Gripper (Present 1 after welding) I181.1/B204.6 RC209/109
            RemoveComponent2Flt : Bool;   // ST1OP09 (WELD HSB2 HV) Remove Component From Gripper (Present 2 after welding) Ixx.X RC225/125
            RemoveComponent3Flt : Bool;   // ST1OP09 (WELD HSB2 HV) Remove Component From Gripper (Present 3 after welding) Ixx.X RC226/126
            RemoveComponent4Flt : Bool;   // ST1OP09 (WELD HSB2 HV) Remove Component From Gripper (Present 4 after welding) Ixx.X RC227/127
            RemoveComponent5Flt : Bool;   // ST1OP09 (WELD HSB2 HV) Remove Component From Gripper (Present 5 after welding) Ixx.X RC228/128
            RemoveComponent6Flt : Bool;   // ST1OP09 (WELD HSB2 HV) Remove Component From Gripper (Present 6 after welding) Ixx.X RC229/129
            RemoveComponent7Flt : Bool;   // ST1OP09 (WELD HSB2 HV) Remove Component From Gripper (Present 7 after welding) Ixx.X RC230/130
            RemoveComponent8Flt : Bool;   // ST1OP09 (WELD HSB2 HV) Remove Component From Gripper (Present 8 after welding) Ixx.X RC231/131
            CompMissing1Flt : Bool;   // ST1OP09 (WELD HSB2 HV) Component Present 1 Missing In Gripper I181.1/B204.6 RC210/110
            CompMissing2Flt : Bool;   // ST1OP09 (WELD HSB2 HV) Component Present 2 Missing In Gripper Ixx.X RC232/132
            CompMissing3Flt : Bool;   // ST1OP09 (WELD HSB2 HV) Component Present 3 Missing In Gripper Ixx.X RC233/133
            CompMissing4Flt : Bool;   // ST1OP09 (WELD HSB2 HV) Component Present 4 Missing In Gripper Ixx.X RC234/134
            CompMissing5Flt : Bool;   // ST1OP09 (WELD HSB2 HV) Component Present 5 Missing In Gripper Ixx.X RC235/135
            CompMissing6Flt : Bool;   // ST1OP09 (WELD HSB2 HV) Component Present 6 Missing In Gripper Ixx.X RC236/136
            CompMissing7Flt : Bool;   // ST1OP09 (WELD HSB2 HV) Component Present 7 Missing In Gripper Ixx.X RC237/137
            CompMissing8Flt : Bool;   // ST1OP09 (WELD HSB2 HV) Component Present 8 Missing In Gripper Ixx.X RC238/138
            SpareFaultRC : Byte;
            HotplateTempOutFlt : Bool;   // ST1OP09 (WELD HSB2 HV) Hotplate Temperature Out Of Tolerance
            HotplateTempSensorFlt : Bool;   // ST1OP09 (WELD HSB2 HV) Hotplate Thermocouple Wire Break
            HotplateTempDiffereneceTooBigFlt : Bool;   // ST1OP09 (WELD HSB2 HV) Hotplate Thermocouples Difference Too Big
            Reserved0_3 : Bool;
            Reserved0_4 : Bool;
            Reserved0_5 : Bool;
            CompStuckOnTankFlt : Bool;   // ST1OP09 (WELD HSB2 HV) Component Stuck On Tank Must reset to Ungrip Component
            TempSetFlt : Bool;   // ST1OP09 (WELD HSB2 HV) Hotplate Tempearture Setpoint Out Of Range
            Reserved1_0 : Bool;
            RemoveHeatedComponentFlt : Bool;   // ST1OP09 (WELD HSB2 HV) Remove Heated Component
            CleanHotplatesFlt : Bool;   // ST1OP09 (WELD HSB2 HV) Clean Hotplates
            NoDetectionUsed : Bool;   // ST1OP09 (WELD HSB2 HV) No Detection Used (PLC program issue)
            SpareAlarmsDInt0 : DInt;
            HotTempChanFlt : Bool;   // ST1OP09 (WELD HSB2 HV) Hotplate Temperature is not changing
            Spare_1 : Bool;
            Spare_2 : Bool;
            Spare_3 : Bool;
            Spare_4 : Bool;
            Spare_5 : Bool;
            TrCommonAdvFlt : Bool;
            TrCommonRetFlt : Bool;
            TrCommonTsFlt : Bool;
            Spare_6 : Bool;
            Spare_7 : Bool;
            Spare_8 : Bool;
            TrStopperVerticalWPAlm : Bool;
            TrStopperVerticalPPAlm : Bool;
            TrStopperVerticalBSAlm : Bool;
            Spare_9 : Bool;
            Spare_10 : Bool;
            Spare_11 : Bool;
            Spare_12 : Bool;
            Spare_13 : Bool;
            Spare_14 : Bool;
            Spare_15 : Bool;
            Spare_16 : Bool;
            Spare_17 : Bool;
            Spare_18 : Bool;
            Spare_19 : Bool;
            Spare_20 : Bool;
            Spare_21 : Bool;
            Spare_22 : Bool;
            Spare_23 : Bool;
            Spare_24 : Bool;
            Spare_25 : Bool;
            Spare_26 : Bool;
            Spare_27 : Bool;
            Spare_28 : Bool;
            Spare_29 : Bool;
            Spare_30 : Bool;
            Spare_31 : Bool;
            Spare_32 : Bool;
            RemCycleNotStartedBADFromPrevStation : Bool;   // ST1OP09 (WELD HSB2 HV) Reminder Cycle Not Started BAD From Previously Station
            Spare_34 : Bool;
         END_STRUCT;
         ST1OP10 : Struct   // WELD / WELD HSB3 HV
            HeaterTransferAdvFlt : Bool;   // ST1OP10 (WELD HSB3 HV) Heater Transfer Failed to Advance Ixx.X
            HeaterTransferRetFlt : Bool;   // ST1OP10 (WELD HSB3 HV) Heater Transfer Failed to Return Ixx.X
            HeaterTransferTSFlt : Bool;   // ST1OP10 (WELD HSB3 HV) Heater Transfer Two Sensors on Ixx.X-Ixx.X
            GcylAdvHeatingFlt : Bool;   // ST1OP10 (WELD HSB3 HV) Gcyl Failed to Advance Heating I110.2/B206.8
            GcylAdvCoolingFlt : Bool;   // ST1OP10 (WELD HSB3 HV) Gcyl Failed to Advance Cooling I110.1/B206.6
            GcylAdvLoadingFlt : Bool;   // ST1OP10 (WELD HSB3 HV) Gcyl Failed to Advance Loading I110.0/B206.4
            GcylRetFlt : Bool;   // ST1OP10 (WELD HSB3 HV) Gcyl Failed to Return I110.3/B206.10
            GcylTSFlt : Bool;   // ST1OP10 (WELD HSB3 HV) Gcyl Two Sensors on I110.0/B206.4 - I110.3/B206.10
            HcylAdvFlt : Bool;   // ST1OP10 (WELD HSB3 HV) Hcyl Failed to Advance I110.4/B206.12 (Ret Sensor for BC)
            HcylRevFlt : Bool;   // ST1OP10 (WELD HSB3 HV) Hcyl Failed to Return I110.5/B206.14
            HcylTSFlt : Bool;   // ST1OP10 (WELD HSB3 HV) Hcyl Two Sensors on I110.4/B206.12-I110.5/B206.14
            GripperAdvGripFlt : Bool;   // ST1OP10 (WELD HSB3 HV) Gripper Failed to Grip (Ungrip sensor Fault) I110.6/B206.16
            GripperRetUngripFlt : Bool;   // ST1OP10 (WELD HSB3 HV) Gripper Failed to Ungrip Sensor Fault I110.6/B206.18
            GripTSFlt : Bool;   // not used
            SpareCylFaultsInt0 : Int;
            SpareCylFaultsDInt0 : DInt;
            CompHeatPosFlt : Bool;   // ST1OP10 (WELD HSB3 HV) Component Failed To Gcyl Heating Position I110.2/B206.8 RC201/101
            TankHeatPosFlt : Bool;   // ST1OP10 (WELD HSB3 HV) Hotplate Failed To Hcyl Heating Position I110.4/B206.12 RC217
            CompCoolPosFlt : Bool;   // ST1OP10 (WELD HSB3 HV) Component Failed To Gcyl Cooling Position I110.1/B206.6 RC202/102
            OpenTimeFlt : Bool;   // ST1OP10 (WELD HSB3 HV) Open Time Exceeded RC203/103
            TempDuringCycleFlt : Bool;   // ST1OP10 (WELD HSB3 HV) Hotplate Temperature Fault During Cycle RC204/104
            ReservedRC0_5 : Bool;
            CompHeatPressFlt : Bool;   // ST1OP10 (WELD HSB3 HV) Component Heating Pressure Out Of Tolerance RC205/105
            ReservedRC0_7 : Bool;
            CompCoolPressFlt : Bool;   // ST1OP10 (WELD HSB3 HV) Component Cooling Pressure Out Of Tolerance RC206/106
            ReservedRC1_1 : Bool;
            ReservedRC1_2 : Bool;
            ReservedRC1_3 : Bool;
            ReservedRC1_4 : Bool;
            ReservedRC1_5 : Bool;
            TankHeatPressFlt : Bool;   // ST1OP10 (WELD HSB3 HV) Hcyl Heating Pressure Out Of Tolerance RC207/107
            ReservedRC1_7 : Bool;
            ReservedRC2_0 : Bool;
            ReservedRC2_1 : Bool;
            ReservedRC2_2 : Bool;
            ReservedRC2_3 : Bool;
            CycleNotFinishFlt : Bool;   // ST1OP10 (WELD HSB3 HV) Cycle Failed To Finish RC211/111
            CycleNotStartedFlt : Bool;   // ST1OP10 (WELD HSB3 HV) Cycle Not Started Fault RC212/112
            ReservedRC2_6 : Bool;
            ReservedRC2_7 : Bool;
            ReservedRC3_0 : Bool;
            TankHeatContactFlt : Bool;   // ST1OP10 (WELD HSB3 HV) Tank Heating Contact Pressure Calc Out Of Tolerance RC213/113
            ReservedRC3_2 : Bool;
            ReservedRC3_3 : Bool;
            MeltedComponentFlt : Bool;   // ST1OP10 (WELD HSB3 HV) Remove Melted Component From Gripper I181.2/B204.8 RC214/114
            ReservedRC3_5 : Bool;
            CylFaultDuringCycleFlt : Bool;   // ST1OP10 (WELD HSB3 HV) Cylinder Fault During Cycle RC215/115
            ReservedRC3_7 : Bool;
            ManualUsedFlt : Bool;   // ST1OP10 (WELD HSB3 HV) Manual Movements Used RC216/116
            CompPresent1AfterHeatFlt : Bool;   // ST1OP10 (WELD HSB3 HV) Component Present 1 Missing After Heating I181.2/B204.8 RC208/108
            CompPresent2AfterHeatFlt : Bool;   // ST1OP10 (WELD HSB3 HV) Component Present 2 Missing After Heating Ixx.X RC218/118
            CompPresent3AfterHeatFlt : Bool;   // ST1OP10 (WELD HSB3 HV) Component Present 3 Missing After Heating Ixx.X RC219/119
            CompPresent4AfterHeatFlt : Bool;   // ST1OP10 (WELD HSB3 HV) Component Present 4 Missing After Heating Ixx.X RC220/120
            CompPresent5AfterHeatFlt : Bool;   // ST1OP10 (WELD HSB3 HV) Component Present 5 Missing After Heating Ixx.X RC221/121
            CompPresent6AfterHeatFlt : Bool;   // ST1OP10 (WELD HSB3 HV) Component Present 6 Missing After Heating Ixx.X RC222/122
            CompPresent7AfterHeatFlt : Bool;   // ST1OP10 (WELD HSB3 HV) Component Present 7 Missing After Heating Ixx.X RC223/123
            CompPresent8AfterHeatFlt : Bool;   // ST1OP10 (WELD HSB3 HV) Component Present 8 Missing After Heating Ixx.X RC224/124
            RemoveComponent1Flt : Bool;   // ST1OP10 (WELD HSB3 HV) Remove Component From Gripper (Present 1 after welding) I181.2/B204.8 RC209/109
            RemoveComponent2Flt : Bool;   // ST1OP10 (WELD HSB3 HV) Remove Component From Gripper (Present 2 after welding) Ixx.X RC225/125
            RemoveComponent3Flt : Bool;   // ST1OP10 (WELD HSB3 HV) Remove Component From Gripper (Present 3 after welding) Ixx.X RC226/126
            RemoveComponent4Flt : Bool;   // ST1OP10 (WELD HSB3 HV) Remove Component From Gripper (Present 4 after welding) Ixx.X RC227/127
            RemoveComponent5Flt : Bool;   // ST1OP10 (WELD HSB3 HV) Remove Component From Gripper (Present 5 after welding) Ixx.X RC228/128
            RemoveComponent6Flt : Bool;   // ST1OP10 (WELD HSB3 HV) Remove Component From Gripper (Present 6 after welding) Ixx.X RC229/129
            RemoveComponent7Flt : Bool;   // ST1OP10 (WELD HSB3 HV) Remove Component From Gripper (Present 7 after welding) Ixx.X RC230/110
            RemoveComponent8Flt : Bool;   // ST1OP10 (WELD HSB3 HV) Remove Component From Gripper (Present 8 after welding) Ixx.X RC231/131
            CompMissing1Flt : Bool;   // ST1OP10 (WELD HSB3 HV) Component Present 1 Missing In Gripper I181.2/B204.8 RC210/110
            CompMissing2Flt : Bool;   // ST1OP10 (WELD HSB3 HV) Component Present 2 Missing In Gripper Ixx.X RC232/132
            CompMissing3Flt : Bool;   // ST1OP10 (WELD HSB3 HV) Component Present 3 Missing In Gripper Ixx.X RC233/133
            CompMissing4Flt : Bool;   // ST1OP10 (WELD HSB3 HV) Component Present 4 Missing In Gripper Ixx.X RC234/134
            CompMissing5Flt : Bool;   // ST1OP10 (WELD HSB3 HV) Component Present 5 Missing In Gripper Ixx.X RC235/135
            CompMissing6Flt : Bool;   // ST1OP10 (WELD HSB3 HV) Component Present 6 Missing In Gripper Ixx.X RC236/136
            CompMissing7Flt : Bool;   // ST1OP10 (WELD HSB3 HV) Component Present 7 Missing In Gripper Ixx.X RC237/137
            CompMissing8Flt : Bool;   // ST1OP10 (WELD HSB3 HV) Component Present 8 Missing In Gripper Ixx.X RC238/138
            SpareFaultRC : Byte;
            HotplateTempOutFlt : Bool;   // ST1OP10 (WELD HSB3 HV) Hotplate Temperature Out Of Tolerance
            HotplateTempSensorFlt : Bool;   // ST1OP10 (WELD HSB3 HV) Hotplate Thermocouple Wire Break
            HotplateTempDiffereneceTooBigFlt : Bool;   // ST1OP10 (WELD HSB3 HV) Hotplate Thermocouples Difference Too Big
            Reserved0_3 : Bool;
            Reserved0_4 : Bool;
            Reserved0_5 : Bool;
            CompStuckOnTankFlt : Bool;   // ST1OP10 (WELD HSB3 HV) Component Stuck On Tank Must reset to Ungrip Component
            TempSetFlt : Bool;   // ST1OP10 (WELD HSB3 HV) Hotplate Tempearture Setpoint Out Of Range
            Reserved1_0 : Bool;
            RemoveHeatedComponentFlt : Bool;   // ST1OP10 (WELD HSB3 HV) Remove Heated Component
            CleanHotplatesFlt : Bool;   // ST1OP10 (WELD HSB3 HV) Clean Hotplates
            NoDetectionUsed : Bool;   // ST1OP10 (WELD HSB3 HV) No Detection Used (PLC program issue)
            SpareAlarmsDInt0 : DInt;
            HotTempChanFlt : Bool;   // ST1OP10 (WELD HSB3 HV) Hotplate Temperature is not changing
            Spare_1 : Bool;
            Spare_2 : Bool;
            Spare_3 : Bool;
            Spare_4 : Bool;
            Spare_5 : Bool;
            TrCommonAdvFlt : Bool;
            TrCommonRetFlt : Bool;
            TrCommonTsFlt : Bool;
            Spare_6 : Bool;
            Spare_7 : Bool;
            Spare_8 : Bool;
            TrStopperVerticalWPAlm : Bool;
            TrStopperVerticalPPAlm : Bool;
            TrStopperVerticalBSAlm : Bool;
            Spare_9 : Bool;
            Spare_10 : Bool;
            Spare_11 : Bool;
            Spare_12 : Bool;
            Spare_13 : Bool;
            Spare_14 : Bool;
            Spare_15 : Bool;
            Spare_16 : Bool;
            Spare_17 : Bool;
            Spare_18 : Bool;
            Spare_19 : Bool;
            Spare_20 : Bool;
            Spare_21 : Bool;
            Spare_22 : Bool;
            Spare_23 : Bool;
            Spare_24 : Bool;
            Spare_25 : Bool;
            Spare_26 : Bool;
            Spare_27 : Bool;
            Spare_28 : Bool;
            Spare_29 : Bool;
            Spare_30 : Bool;
            Spare_31 : Bool;
            Spare_32 : Bool;
            RemCycleNotStartedBADFromPrevStation : Bool;   // ST1OP10 (WELD HSB3 HV) Reminder Cycle Not Started BAD From Previously Station
            Spare_34 : Bool;
         END_STRUCT;
         ST1OP11 : Struct   // DESTROYER
            TransferWPAlm : Bool;   // ST1OP11 (DESTROYER) Drilling transfer failed to advance I121.4/B177.12
            TransferPPAlm : Bool;   // ST1OP11 (DESTROYER) Drilling transfer failed to reverse I121.5/B177.14
            TransferBSAlm : Bool;   // ST1OP11 (DESTROYER) Drilling transfer both sensors ON I121.4-5/B177.12-14
            DrillMissing : Bool;   // ST1OP11 (DESTROYER) Drill missing I121.6/B177.16
            Spare_0_4 : Bool;
            Spare_0_5 : Bool;
            Spare_0_6 : Bool;
            Spare_0_7 : Bool;
            Spare_1_0 : Bool;
            Spare_1_1 : Bool;
            Spare_1_2 : Bool;
            Spare_1_3 : Bool;
            Spare_1_4 : Bool;
            Spare_1_5 : Bool;
            Spare_1_6 : Bool;
            Spare_1_7 : Bool;
            Temp1 : Array[2..9] of Byte;
         END_STRUCT;
         Spare : Array[80..99] of Byte;
      END_STRUCT;
      ST2 : Struct
         GENERAL : Struct   // GENERAL ST2
            TankBAD : Bool;   // Tank BAD after Manual Mode
            VerCrossed : Bool;   // ST2 Vertical light curtain crossed without authorization
            HorCrossed : Bool;   // ST2 Horizontal light curtain crossed without authorization
            VerNotEngaged : Bool;   // ST2 Cannot engage vertical light curtain
            HorNotEngaged : Bool;   // ST2 Cannot engage horizontal light curtain
            VerActive : Bool;   // ST2 Vertical light curtain not active
            HorActive : Bool;   // ST2 Horizontal light curtain not active
            TankAbsent_FOTO : Bool;   // ST2 Tank absent on foto I201.2/B275.8
            Tank_TempOutOfTol : Bool;   // Tank temperature out of tolerance PIW500 / B190.3
            Tank_TempSensBrok : Bool;   // Tank temperature sensor broken PIW500 / B190.3
            SqlST1 : Bool;   // ST2 SQL Trigger not reseted after 10s
            SqlST2 : Bool;   // ST3 SQL Trigger not reseted after 10s
            SqlST3 : Bool;   // ST4 SQL Trigger not reseted after 10s
            SqlST4 : Bool;   // ST1 SQL Trigger not reseted after 10s
            TankAbsent_ISOPIN_L : Bool;   // ST2 Tank absent on ISOPIN Left I200.0/B274.4
            TankAbsent_ISOPIN_R : Bool;   // ST2 Tank absent on ISOPIN Right I200.1/B274.6
            BarcodeTankNotRead : Bool;   // Alarm Tank barcode not read
            BarcodeTankNotCorrect : Bool;   // Alarm Tank barcode not correct with selected version
            FIFO_Tank : Bool;   // FIFO Alarm - Tank was processed
            Spare2_3 : Bool;
            BarcodeTankNotRead2 : Bool;   // Alarm Tank barcode 2not read
            BarcodeTankNotCorrect2 : Bool;   // Alarm Tank barcode2 not correct with selected version
            FIFO_Tank2 : Bool;   // FIFO Alarm 2- Tank was processed
            Spare2_7 : Bool;
            NoReleaseToStart : Bool;   // No release authorization from Traceability for Station 1 start cycle. Please acknowledge.
            NoReleaseToUnclamp : Bool;   // No release authorization from Traceability for Station 1 unclamp Tank. Please acknowledge.
            WaitReletoStAlmRes : Bool;   // Traceability for Station 1 is waiting for release to start alarm reset
            WaitResultReadAlmRes : Bool;   // Traceability for Station 1 is waiting for result read alarm reset
            TraceTrigON : Bool;   // Station 1 Traceability log fault (trigger still ON)
            Spare3_5 : Bool;
            Spare3_6 : Bool;
            Spare3_7 : Bool;
            TableDobulPos : Bool;   // Table double position fault
            TableInvertNotEn : Bool;   // Fault Tank temperature out of tolerance / Table Inverter not enable
            TablerInvNotReady : Bool;   // Fault Tank temperature sensor broken / Table inverter not ready
            TableNotInPos : Bool;   // Empty the slug bin ST1OP1/ST1OP2 / Table indexer not in position
            TableTime : Bool;   // Table timeout fault
            TablePosRun : Bool;   // Table position run over fault
            TableSafety : Bool;   // Table safety fault
            TableSumEr : Bool;   // ST1OP01 CUT FSU Slug not detected frame I120.4/B157.10 / Table Sum error
            TableSumWar : Bool;   // ST1OP02 CUT ICV Slug not detected frame I120.3/B157.12 / Table sum warning
            Spare5_1 : Bool;
            Spare5_2 : Bool;
            ST1PunchingBoxFull : Bool;
            spare_1 : Bool;
            TankWithoutStatusFromPrevST : Bool;   // Tube without any status on Station 1. Impossible to proceed with this Tube
            TankNotInFIFO : Bool;   // Tank not in FIFO. Impossible to proceed with this Tube
            TankWithBADStatusFromPrevST : Bool;   // Tank Status BAD on Station ST1. Tank will be destroyed. Press START
            Spare : Array[6..9] of Byte;
         END_STRUCT;
         SidoorFront : Struct
            "DoorFrontSidorAl-1" : Bool;   // ST2 Door sidoor Front - RAM, EEPROM or CPU error (system error)
            "DoorFrontSidorAl-2" : Bool;   // ST2 Door sidoor Front - Braking chopper defective
            "DoorFrontSidorAl-3" : Bool;   // ST2 Door sidoor Front - Error in the second shutdown route
            "DoorFrontSidorAl-4" : Bool;   // ST2 Door sidoor Front - Motor protection, maximum opening or closing time of 65 s has been exceeded
            "DoorFrontSidorAl-5" : Bool;   // ST2 Door sidoor Front - Motor undefined – no learn run carried out with this motor type (If a different motor version is used, the learn run must be repeated at power on as described in these Operating
            "DoorFrontSidorAl-6" : Bool;   // ST2 Door sidoor Front -
            "DoorFrontSidorAl-7" : Bool;   // ST2 Door sidoor Front - Error in pulse generator
            "DoorFrontSidorAl-8" : Bool;   // ST2 Door sidoor Front - OSSD (ESPE type 2 or pressure-sensitive edge) – Function test failed
            "DoorFrontSidorAl-9" : Bool;   // ST2 Door sidoor Front - Motor overcurrent
            "DoorFrontSidorAl-E" : Bool;   // ST2 Door sidoor Front - Motor overvoltage
            "DoorFrontSidorAl-F" : Bool;   // ST2 Door sidoor Front - Motor undervoltage
            "DoorFrontSidorAl-n" : Bool;   // ST2 Door sidoor Front - Output stage defective
            "DoorFrontSidorAl-L" : Bool;   // ST2 Door sidoor Front - Current measurement error
            "DoorFrontSidorAl-t" : Bool;   // ST2 Door sidoor Front - Belt torn
            "DoorFrontSidorAl-U" : Bool;   // ST2 Door sidoor Front - Max. mass to be moved:
            "Spare 1_7" : Bool;
            CloseDoorByHand : Bool;   // ST2 Door sidoor Front - close by hand
            DoorFrontLearn : Bool;   // ST2 Doors front in learn procedure - Please Wait
            DoorFrontSpecial : Bool;   // Please Wait - Sidoor Front in Special - mode The system is in an error state or special mode (system is shutting down, powering up or saving safety-related parameters)
            SidoorFrontOpenAlarm : Bool;   // Sidoor Front - An obstruction was detected in the opening direction
            SidoorFrontCloseAlarm : Bool;   // Sidoor Front - An obstruction was detected in the closing direction
            Temp1 : Array[4..9] of Byte;
         END_STRUCT;
         SidoorSide : Struct
            "DoorSideSidorAl-1" : Bool;   // ST2 Door sidoor Side - RAM, EEPROM or CPU error (system error)
            "DoorSideSidorAl-2" : Bool;   // ST2 Door sidoor Side - Braking chopper defective
            "DoorSideSidorAl-3" : Bool;   // ST2 Door sidoor Side - Error in the second shutdown route
            "DoorSideSidorAl-4" : Bool;   // ST2 Door sidoor Side - Motor protection, maximum opening or closing time of 65 s has been exceeded
            "DoorSideSidorAl-5" : Bool;   // ST2 Door sidoor Side - Motor undefined – no learn run carried out with this motor type (If a different motor version is used, the learn run must be repeated at power on as described in these Operating
            "DoorSideSidorAl-6" : Bool;   // ST2 Door sidoor Side -
            "DoorSideSidorAl-7" : Bool;   // ST2 Door sidoor Side - Error in pulse generator
            "DoorSideSidorAl-8" : Bool;   // ST2 Door sidoor Side - OSSD (ESPE type 2 or pressure-sensitive edge) – Function test failed
            "DoorSideSidorAl-9" : Bool;   // ST2 Door sidoor Side - Motor overcurrent
            "DoorSideSidorAl-E" : Bool;   // ST2 Door sidoor Side - Motor overvoltage
            "DoorSideSidorAl-F" : Bool;   // ST2 Door sidoor Side - Motor undervoltage
